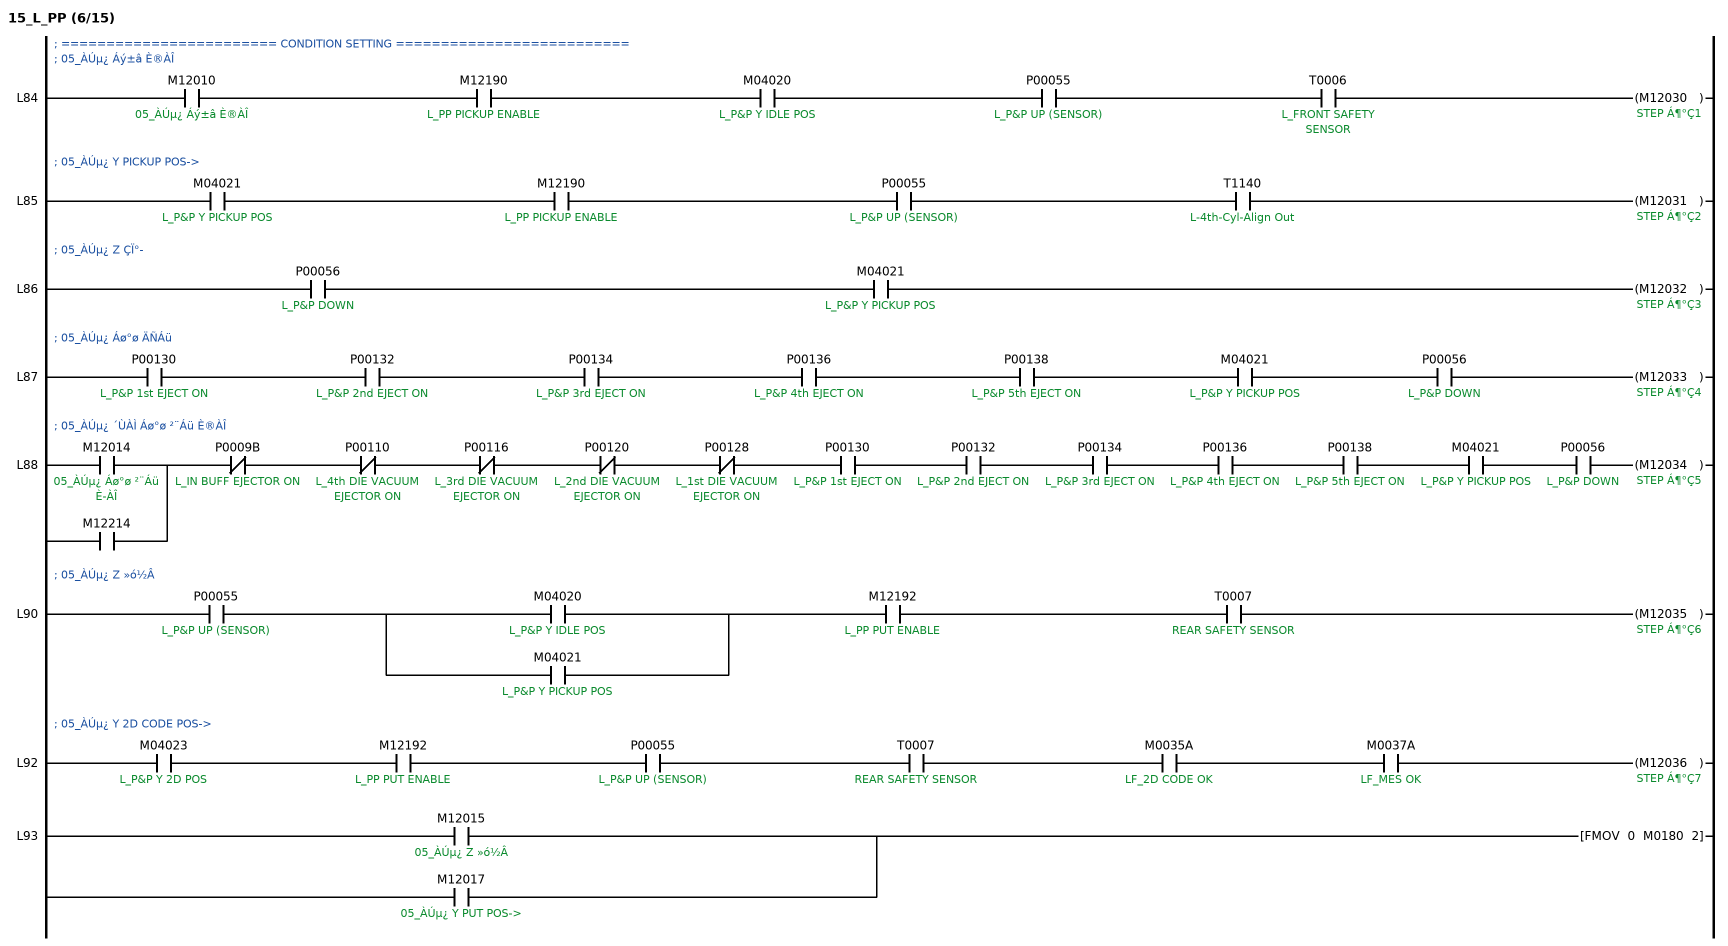
[picture p120: 15_L_PP rungs L84-L93]
// ======================== CONDITION SETTING ==========================
; L84
LOAD      M12010	// 05_ÀÚµ¿ Áý±â È®ÀÎ
AND       M12190	// L_PP PICKUP ENABLE
AND       M04020	// L_P&P Y IDLE POS
AND       P00055	// L_P&P UP (SENSOR)
AND       T0006	// L_FRONT SAFETY SENSOR
OUT       M12030	// STEP Á¶°Ç1
// output comment: 05_ÀÚµ¿ Áý±â È®ÀÎ
; L85
LOAD      M04021	// L_P&P Y PICKUP POS
AND       M12190	// L_PP PICKUP ENABLE
AND       P00055	// L_P&P UP (SENSOR)
AND       T1140	// L-4th-Cyl-Align Out
OUT       M12031	// STEP Á¶°Ç2
// output comment: 05_ÀÚµ¿ Y PICKUP POS->
; L86
LOAD      P00056	// L_P&P DOWN
AND       M04021	// L_P&P Y PICKUP POS
OUT       M12032	// STEP Á¶°Ç3
// output comment: 05_ÀÚµ¿ Z ÇÏ°­
; L87
LOAD      P00130	// L_P&P 1st EJECT ON
AND       P00132	// L_P&P 2nd EJECT ON
AND       P00134	// L_P&P 3rd EJECT ON
AND       P00136	// L_P&P 4th EJECT ON
AND       P00138	// L_P&P 5th EJECT ON
AND       M04021	// L_P&P Y PICKUP POS
AND       P00056	// L_P&P DOWN
OUT       M12033	// STEP Á¶°Ç4
// output comment: 05_ÀÚµ¿ Áø°ø ÄÑÁü
; L88
LOAD      M12014	// 05_ÀÚµ¿ Áø°ø ²¨Áü È­ÀÎ
OR        M12214
AND NOT   P0009B	// L_IN BUFF EJECTOR ON
AND NOT   P00110	// L_4th DIE VACUUM EJECTOR ON
AND NOT   P00116	// L_3rd DIE VACUUM EJECTOR ON
AND NOT   P00120	// L_2nd DIE VACUUM EJECTOR ON
AND NOT   P00128	// L_1st DIE VACUUM EJECTOR ON
AND       P00130	// L_P&P 1st EJECT ON
AND       P00132	// L_P&P 2nd EJECT ON
AND       P00134	// L_P&P 3rd EJECT ON
AND       P00136	// L_P&P 4th EJECT ON
AND       P00138	// L_P&P 5th EJECT ON
AND       M04021	// L_P&P Y PICKUP POS
AND       P00056	// L_P&P DOWN
OUT       M12034	// STEP Á¶°Ç5
// output comment: 05_ÀÚµ¿ ´ÙÀÌ Áø°ø ²¨Áü È®ÀÎ
; L90
LOAD      P00055	// L_P&P UP (SENSOR)
LOAD      M04020	// L_P&P Y IDLE POS
OR        M04021	// L_P&P Y PICKUP POS
AND LOAD
AND       M12192	// L_PP PUT ENABLE
AND       T0007	// REAR SAFETY SENSOR
OUT       M12035	// STEP Á¶°Ç6
// output comment: 05_ÀÚµ¿ Z »ó½Â
; L92
LOAD      M04023	// L_P&P Y 2D POS
AND       M12192	// L_PP PUT ENABLE
AND       P00055	// L_P&P UP (SENSOR)
AND       T0007	// REAR SAFETY SENSOR
AND       M0035A	// LF_2D CODE OK
AND       M0037A	// LF_MES OK
OUT       M12036	// STEP Á¶°Ç7
// output comment: 05_ÀÚµ¿ Y 2D CODE POS->
; L93
LOAD      M12015	// 05_ÀÚµ¿ Z »ó½Â
OR        M12017	// 05_ÀÚµ¿ Y PUT POS->
FMOV      0 M0180 2

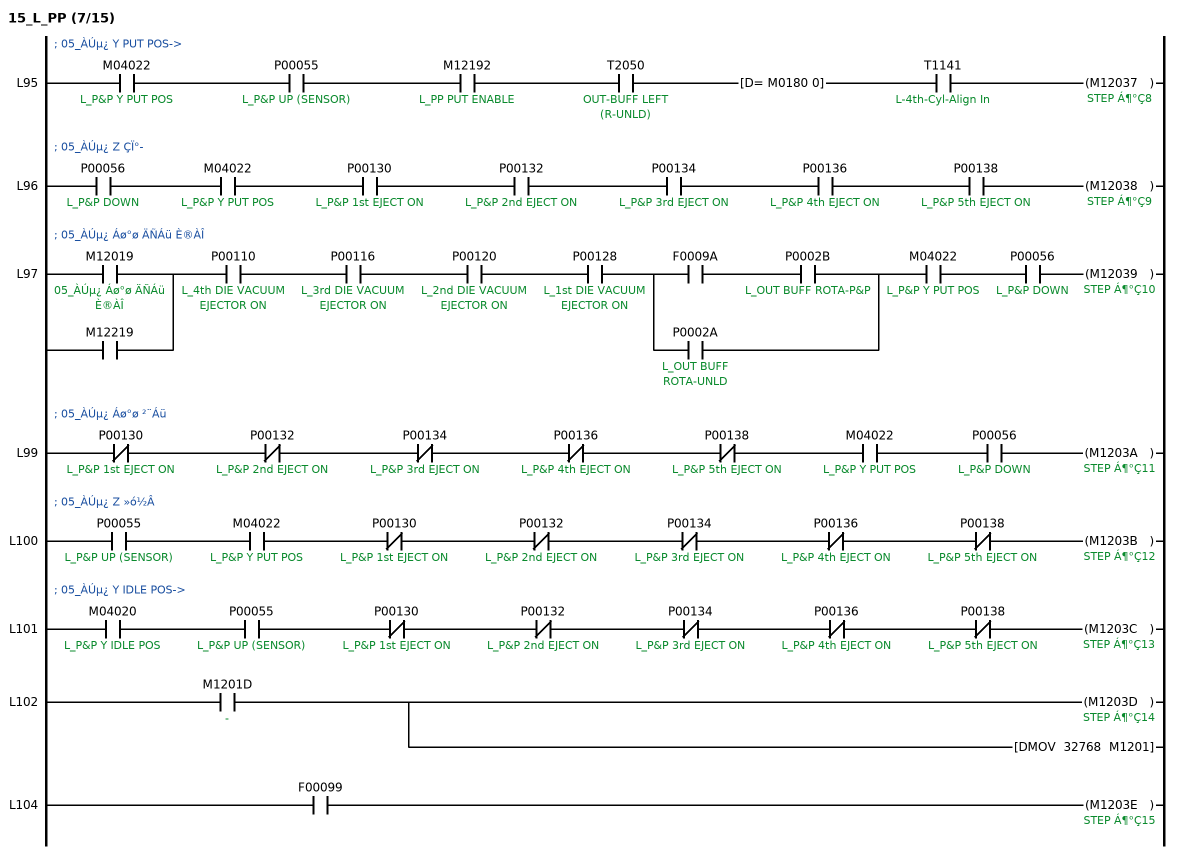
; L95
LOAD      M04022	// L_P&P Y PUT POS
AND       P00055	// L_P&P UP (SENSOR)
AND       M12192	// L_PP PUT ENABLE
AND       T2050	// OUT-BUFF LEFT (R-UNLD)
ANDD=     M0180 0
AND       T1141	// L-4th-Cyl-Align In
OUT       M12037	// STEP Á¶°Ç8
// output comment: 05_ÀÚµ¿ Y PUT POS->
; L96
LOAD      P00056	// L_P&P DOWN
AND       M04022	// L_P&P Y PUT POS
AND       P00130	// L_P&P 1st EJECT ON
AND       P00132	// L_P&P 2nd EJECT ON
AND       P00134	// L_P&P 3rd EJECT ON
AND       P00136	// L_P&P 4th EJECT ON
AND       P00138	// L_P&P 5th EJECT ON
OUT       M12038	// STEP Á¶°Ç9
// output comment: 05_ÀÚµ¿ Z ÇÏ°­
; L97
LOAD      M12019	// 05_ÀÚµ¿ Áø°ø ÄÑÁü È®ÀÎ
OR        M12219
AND       P00110	// L_4th DIE VACUUM EJECTOR ON
AND       P00116	// L_3rd DIE VACUUM EJECTOR ON
AND       P00120	// L_2nd DIE VACUUM EJECTOR ON
AND       P00128	// L_1st DIE VACUUM EJECTOR ON
LOAD      F0009A
AND       P0002B	// L_OUT BUFF ROTA-P&P
OR        P0002A	// L_OUT BUFF ROTA-UNLD
AND LOAD
AND       M04022	// L_P&P Y PUT POS
AND       P00056	// L_P&P DOWN
OUT       M12039	// STEP Á¶°Ç10
// output comment: 05_ÀÚµ¿ Áø°ø ÄÑÁü È®ÀÎ
; L99
LOAD NOT  P00130	// L_P&P 1st EJECT ON
AND NOT   P00132	// L_P&P 2nd EJECT ON
AND NOT   P00134	// L_P&P 3rd EJECT ON
AND NOT   P00136	// L_P&P 4th EJECT ON
AND NOT   P00138	// L_P&P 5th EJECT ON
AND       M04022	// L_P&P Y PUT POS
AND       P00056	// L_P&P DOWN
OUT       M1203A	// STEP Á¶°Ç11
// output comment: 05_ÀÚµ¿ Áø°ø ²¨Áü
; L100
LOAD      P00055	// L_P&P UP (SENSOR)
AND       M04022	// L_P&P Y PUT POS
AND NOT   P00130	// L_P&P 1st EJECT ON
AND NOT   P00132	// L_P&P 2nd EJECT ON
AND NOT   P00134	// L_P&P 3rd EJECT ON
AND NOT   P00136	// L_P&P 4th EJECT ON
AND NOT   P00138	// L_P&P 5th EJECT ON
OUT       M1203B	// STEP Á¶°Ç12
// output comment: 05_ÀÚµ¿ Z »ó½Â
; L101
LOAD      M04020	// L_P&P Y IDLE POS
AND       P00055	// L_P&P UP (SENSOR)
AND NOT   P00130	// L_P&P 1st EJECT ON
AND NOT   P00132	// L_P&P 2nd EJECT ON
AND NOT   P00134	// L_P&P 3rd EJECT ON
AND NOT   P00136	// L_P&P 4th EJECT ON
AND NOT   P00138	// L_P&P 5th EJECT ON
OUT       M1203C	// STEP Á¶°Ç13
// output comment: 05_ÀÚµ¿ Y IDLE POS->
; L102
LOAD      M1201D	// -
OUT       M1203D	// STEP Á¶°Ç14
DMOV      32768 M1201
; L104
LOAD      F00099
OUT       M1203E	// STEP Á¶°Ç15

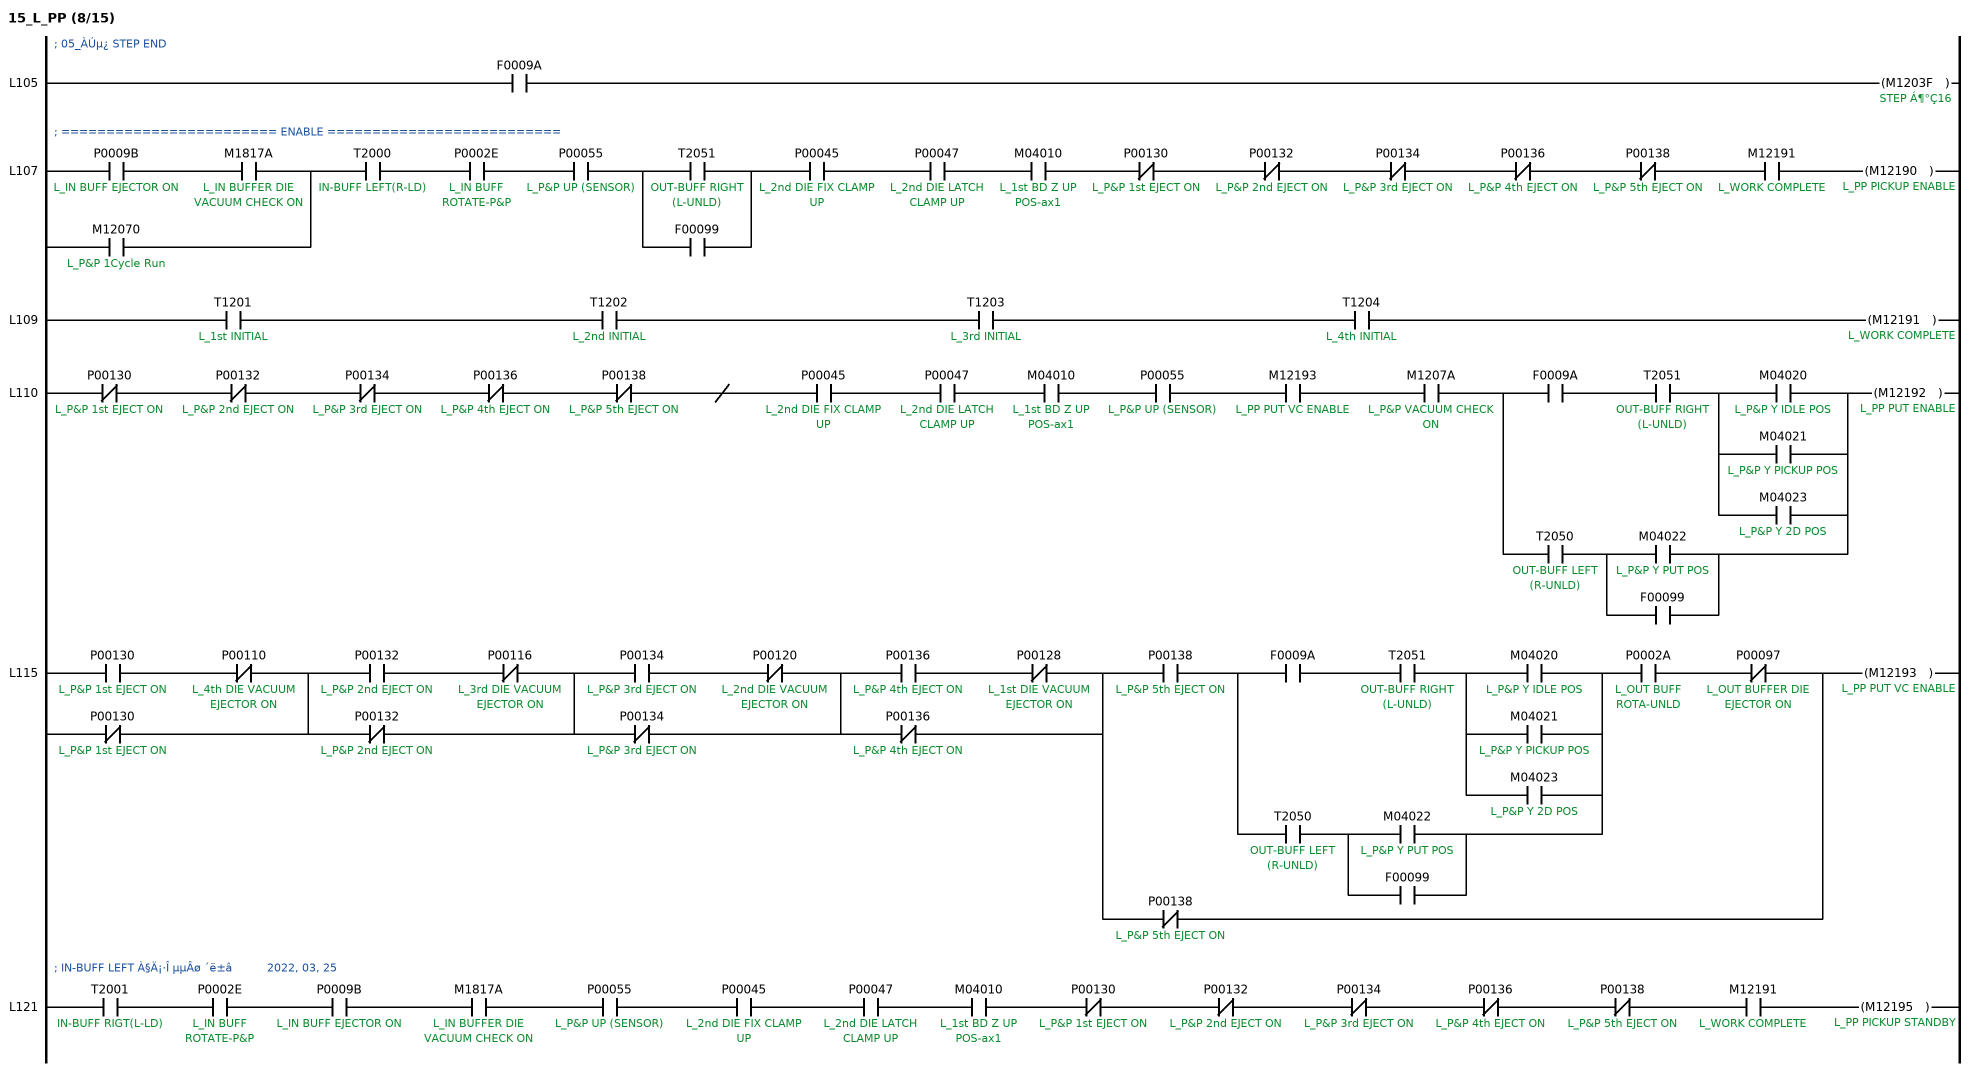
; L105
LOAD      F0009A
OUT       M1203F	// STEP Á¶°Ç16
// output comment: 05_ÀÚµ¿ STEP END
// ======================== ENABLE ==========================
; L107
LOAD      P0009B	// L_IN BUFF EJECTOR ON
AND       M1817A	// L_IN BUFFER DIE VACUUM CHECK ON
OR        M12070	// L_P&P 1Cycle Run
AND       T2000	// IN-BUFF LEFT(R-LD)
AND       P0002E	// L_IN BUFF ROTATE-P&P
AND       P00055	// L_P&P UP (SENSOR)
LOAD      T2051	// OUT-BUFF RIGHT (L-UNLD)
OR        F00099
AND LOAD
AND       P00045	// L_2nd DIE FIX CLAMP UP
AND       P00047	// L_2nd DIE LATCH CLAMP UP
AND       M04010	// L_1st BD Z UP POS-ax1
AND NOT   P00130	// L_P&P 1st EJECT ON
AND NOT   P00132	// L_P&P 2nd EJECT ON
AND NOT   P00134	// L_P&P 3rd EJECT ON
AND NOT   P00136	// L_P&P 4th EJECT ON
AND NOT   P00138	// L_P&P 5th EJECT ON
AND       M12191	// L_WORK COMPLETE
OUT       M12190	// L_PP PICKUP ENABLE
; L109
LOAD      T1201	// L_1st INITIAL
AND       T1202	// L_2nd INITIAL
AND       T1203	// L_3rd INITIAL
AND       T1204	// L_4th INITIAL
OUT       M12191	// L_WORK COMPLETE
; L110
LOAD NOT  P00130	// L_P&P 1st EJECT ON
AND NOT   P00132	// L_P&P 2nd EJECT ON
AND NOT   P00134	// L_P&P 3rd EJECT ON
AND NOT   P00136	// L_P&P 4th EJECT ON
AND NOT   P00138	// L_P&P 5th EJECT ON
NOT
AND       P00045	// L_2nd DIE FIX CLAMP UP
AND       P00047	// L_2nd DIE LATCH CLAMP UP
AND       M04010	// L_1st BD Z UP POS-ax1
AND       P00055	// L_P&P UP (SENSOR)
AND       M12193	// L_PP PUT VC ENABLE
AND       M1207A	// L_P&P VACUUM CHECK ON
LOAD      F0009A
AND       T2051	// OUT-BUFF RIGHT (L-UNLD)
LOAD      M04020	// L_P&P Y IDLE POS
OR        M04021	// L_P&P Y PICKUP POS
OR        M04023	// L_P&P Y 2D POS
AND LOAD
LOAD      T2050	// OUT-BUFF LEFT (R-UNLD)
LOAD      M04022	// L_P&P Y PUT POS
OR        F00099
AND LOAD
OR LOAD
AND LOAD
OUT       M12192	// L_PP PUT ENABLE
; L115
LOAD      P00130	// L_P&P 1st EJECT ON
AND NOT   P00110	// L_4th DIE VACUUM EJECTOR ON
OR NOT    P00130	// L_P&P 1st EJECT ON
LOAD      P00132	// L_P&P 2nd EJECT ON
AND NOT   P00116	// L_3rd DIE VACUUM EJECTOR ON
OR NOT    P00132	// L_P&P 2nd EJECT ON
AND LOAD
LOAD      P00134	// L_P&P 3rd EJECT ON
AND NOT   P00120	// L_2nd DIE VACUUM EJECTOR ON
OR NOT    P00134	// L_P&P 3rd EJECT ON
AND LOAD
LOAD      P00136	// L_P&P 4th EJECT ON
AND NOT   P00128	// L_1st DIE VACUUM EJECTOR ON
OR NOT    P00136	// L_P&P 4th EJECT ON
AND LOAD
LOAD      P00138	// L_P&P 5th EJECT ON
LOAD      F0009A
AND       T2051	// OUT-BUFF RIGHT (L-UNLD)
LOAD      M04020	// L_P&P Y IDLE POS
OR        M04021	// L_P&P Y PICKUP POS
OR        M04023	// L_P&P Y 2D POS
AND LOAD
LOAD      T2050	// OUT-BUFF LEFT (R-UNLD)
LOAD      M04022	// L_P&P Y PUT POS
OR        F00099
AND LOAD
OR LOAD
AND LOAD
AND       P0002A	// L_OUT BUFF ROTA-UNLD
AND NOT   P00097	// L_OUT BUFFER DIE EJECTOR ON
OR NOT    P00138	// L_P&P 5th EJECT ON
AND LOAD
OUT       M12193	// L_PP PUT VC ENABLE
; L121
LOAD      T2001	// IN-BUFF RIGT(L-LD)
AND       P0002E	// L_IN BUFF ROTATE-P&P
AND       P0009B	// L_IN BUFF EJECTOR ON
AND       M1817A	// L_IN BUFFER DIE VACUUM CHECK ON
AND       P00055	// L_P&P UP (SENSOR)
AND       P00045	// L_2nd DIE FIX CLAMP UP
AND       P00047	// L_2nd DIE LATCH CLAMP UP
AND       M04010	// L_1st BD Z UP POS-ax1
AND NOT   P00130	// L_P&P 1st EJECT ON
AND NOT   P00132	// L_P&P 2nd EJECT ON
AND NOT   P00134	// L_P&P 3rd EJECT ON
AND NOT   P00136	// L_P&P 4th EJECT ON
AND NOT   P00138	// L_P&P 5th EJECT ON
AND       M12191	// L_WORK COMPLETE
OUT       M12195	// L_PP PICKUP STANDBY
// output comment: IN-BUFF LEFT À§Ä¡·Î µµÂø ´ë±â          2022, 03, 25

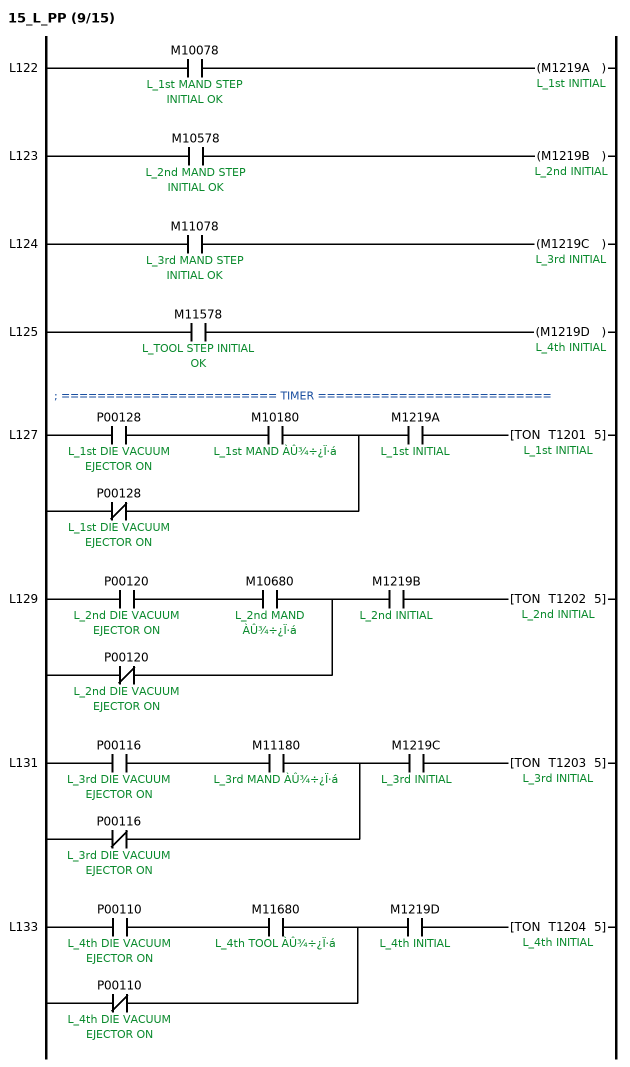
; L122
LOAD      M10078	// L_1st MAND STEP INITIAL OK
OUT       M1219A	// L_1st INITIAL
; L123
LOAD      M10578	// L_2nd MAND STEP INITIAL OK
OUT       M1219B	// L_2nd INITIAL
; L124
LOAD      M11078	// L_3rd MAND STEP INITIAL OK
OUT       M1219C	// L_3rd INITIAL
; L125
LOAD      M11578	// L_TOOL STEP INITIAL OK
OUT       M1219D	// L_4th INITIAL
// ======================== TIMER ==========================
; L127
LOAD      P00128	// L_1st DIE VACUUM EJECTOR ON
AND       M10180	// L_1st MAND ÀÛ¾÷¿Ï·á
OR NOT    P00128	// L_1st DIE VACUUM EJECTOR ON
AND       M1219A	// L_1st INITIAL
TON       T1201 5	// L_1st INITIAL
; L129
LOAD      P00120	// L_2nd DIE VACUUM EJECTOR ON
AND       M10680	// L_2nd MAND ÀÛ¾÷¿Ï·á
OR NOT    P00120	// L_2nd DIE VACUUM EJECTOR ON
AND       M1219B	// L_2nd INITIAL
TON       T1202 5	// L_2nd INITIAL
; L131
LOAD      P00116	// L_3rd DIE VACUUM EJECTOR ON
AND       M11180	// L_3rd MAND ÀÛ¾÷¿Ï·á
OR NOT    P00116	// L_3rd DIE VACUUM EJECTOR ON
AND       M1219C	// L_3rd INITIAL
TON       T1203 5	// L_3rd INITIAL
; L133
LOAD      P00110	// L_4th DIE VACUUM EJECTOR ON
AND       M11680	// L_4th TOOL ÀÛ¾÷¿Ï·á
OR NOT    P00110	// L_4th DIE VACUUM EJECTOR ON
AND       M1219D	// L_4th INITIAL
TON       T1204 5	// L_4th INITIAL

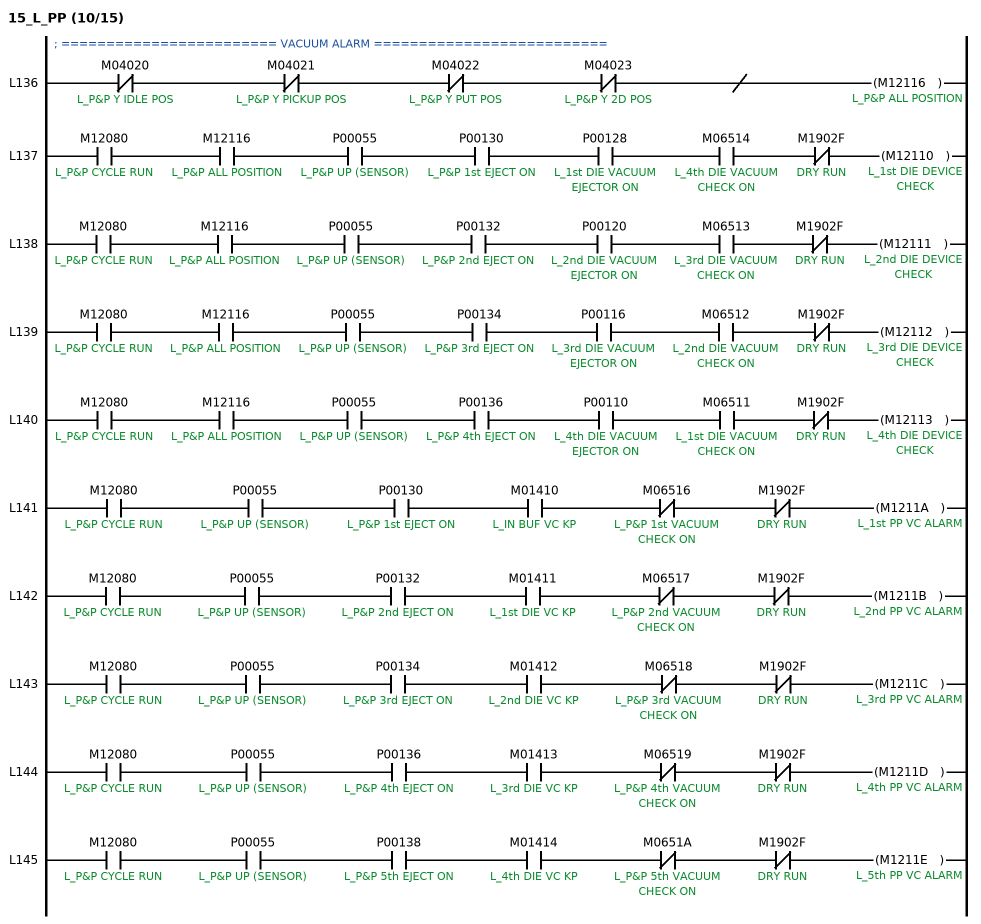
// ======================== VACUUM ALARM ==========================
; L136
LOAD NOT  M04020	// L_P&P Y IDLE POS
AND NOT   M04021	// L_P&P Y PICKUP POS
AND NOT   M04022	// L_P&P Y PUT POS
AND NOT   M04023	// L_P&P Y 2D POS
NOT
OUT       M12116	// L_P&P ALL POSITION
; L137
LOAD      M12080	// L_P&P CYCLE RUN
AND       M12116	// L_P&P ALL POSITION
AND       P00055	// L_P&P UP (SENSOR)
AND       P00130	// L_P&P 1st EJECT ON
AND       P00128	// L_1st DIE VACUUM EJECTOR ON
AND       M06514	// L_4th DIE VACUUM CHECK ON
AND NOT   M1902F	// DRY RUN
OUT       M12110	// L_1st DIE DEVICE CHECK
; L138
LOAD      M12080	// L_P&P CYCLE RUN
AND       M12116	// L_P&P ALL POSITION
AND       P00055	// L_P&P UP (SENSOR)
AND       P00132	// L_P&P 2nd EJECT ON
AND       P00120	// L_2nd DIE VACUUM EJECTOR ON
AND       M06513	// L_3rd DIE VACUUM CHECK ON
AND NOT   M1902F	// DRY RUN
OUT       M12111	// L_2nd DIE DEVICE CHECK
; L139
LOAD      M12080	// L_P&P CYCLE RUN
AND       M12116	// L_P&P ALL POSITION
AND       P00055	// L_P&P UP (SENSOR)
AND       P00134	// L_P&P 3rd EJECT ON
AND       P00116	// L_3rd DIE VACUUM EJECTOR ON
AND       M06512	// L_2nd DIE VACUUM CHECK ON
AND NOT   M1902F	// DRY RUN
OUT       M12112	// L_3rd DIE DEVICE CHECK
; L140
LOAD      M12080	// L_P&P CYCLE RUN
AND       M12116	// L_P&P ALL POSITION
AND       P00055	// L_P&P UP (SENSOR)
AND       P00136	// L_P&P 4th EJECT ON
AND       P00110	// L_4th DIE VACUUM EJECTOR ON
AND       M06511	// L_1st DIE VACUUM CHECK ON
AND NOT   M1902F	// DRY RUN
OUT       M12113	// L_4th DIE DEVICE CHECK
; L141
LOAD      M12080	// L_P&P CYCLE RUN
AND       P00055	// L_P&P UP (SENSOR)
AND       P00130	// L_P&P 1st EJECT ON
AND       M01410	// L_IN BUF VC KP
AND NOT   M06516	// L_P&P 1st VACUUM CHECK ON
AND NOT   M1902F	// DRY RUN
OUT       M1211A	// L_1st PP VC ALARM
; L142
LOAD      M12080	// L_P&P CYCLE RUN
AND       P00055	// L_P&P UP (SENSOR)
AND       P00132	// L_P&P 2nd EJECT ON
AND       M01411	// L_1st DIE VC KP
AND NOT   M06517	// L_P&P 2nd VACUUM CHECK ON
AND NOT   M1902F	// DRY RUN
OUT       M1211B	// L_2nd PP VC ALARM
; L143
LOAD      M12080	// L_P&P CYCLE RUN
AND       P00055	// L_P&P UP (SENSOR)
AND       P00134	// L_P&P 3rd EJECT ON
AND       M01412	// L_2nd DIE VC KP
AND NOT   M06518	// L_P&P 3rd VACUUM CHECK ON
AND NOT   M1902F	// DRY RUN
OUT       M1211C	// L_3rd PP VC ALARM
; L144
LOAD      M12080	// L_P&P CYCLE RUN
AND       P00055	// L_P&P UP (SENSOR)
AND       P00136	// L_P&P 4th EJECT ON
AND       M01413	// L_3rd DIE VC KP
AND NOT   M06519	// L_P&P 4th VACUUM CHECK ON
AND NOT   M1902F	// DRY RUN
OUT       M1211D	// L_4th PP VC ALARM
; L145
LOAD      M12080	// L_P&P CYCLE RUN
AND       P00055	// L_P&P UP (SENSOR)
AND       P00138	// L_P&P 5th EJECT ON
AND       M01414	// L_4th DIE VC KP
AND NOT   M0651A	// L_P&P 5th VACUUM CHECK ON
AND NOT   M1902F	// DRY RUN
OUT       M1211E	// L_5th PP VC ALARM

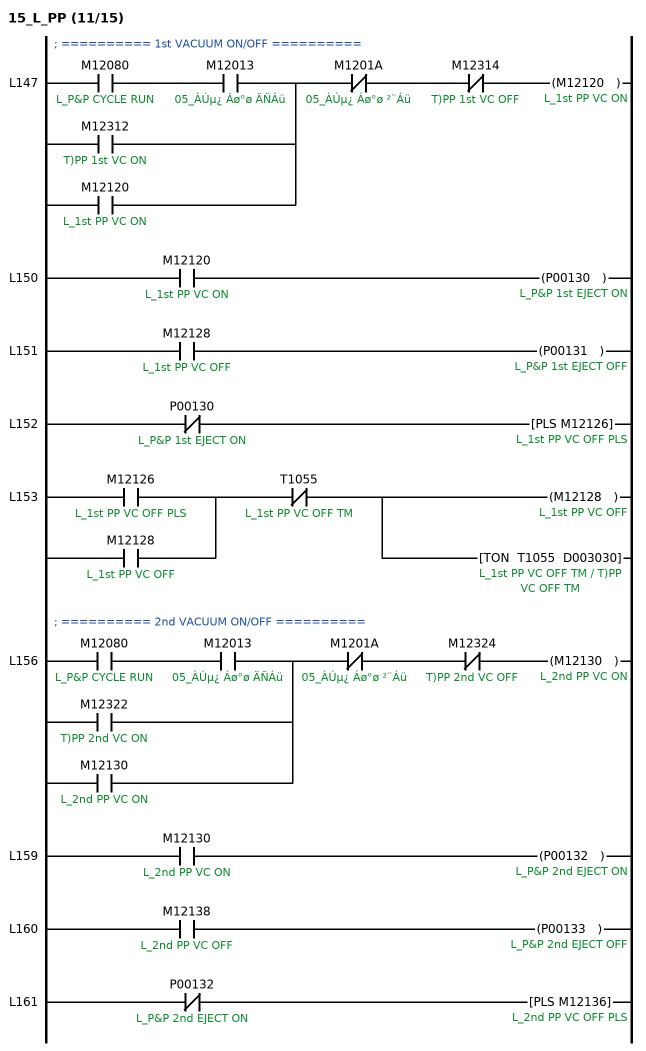
// ========== 1st VACUUM ON/OFF ==========
; L147
LOAD      M12080	// L_P&P CYCLE RUN
AND       M12013	// 05_ÀÚµ¿ Áø°ø ÄÑÁü
OR        M12312	// T)PP 1st VC ON
OR        M12120	// L_1st PP VC ON
AND NOT   M1201A	// 05_ÀÚµ¿ Áø°ø ²¨Áü
AND NOT   M12314	// T)PP 1st VC OFF
OUT       M12120	// L_1st PP VC ON
; L150
LOAD      M12120	// L_1st PP VC ON
OUT       P00130	// L_P&P 1st EJECT ON
; L151
LOAD      M12128	// L_1st PP VC OFF
OUT       P00131	// L_P&P 1st EJECT OFF
; L152
LOAD NOT  P00130	// L_P&P 1st EJECT ON
OUTP      M12126	// L_1st PP VC OFF PLS
; L153
LOAD      M12126	// L_1st PP VC OFF PLS
OR        M12128	// L_1st PP VC OFF
AND NOT   T1055	// L_1st PP VC OFF TM
OUT       M12128	// L_1st PP VC OFF
TON       T1055 D003030	// L_1st PP VC OFF TM / T)PP VC OFF TM
// ========== 2nd VACUUM ON/OFF ==========
; L156
LOAD      M12080	// L_P&P CYCLE RUN
AND       M12013	// 05_ÀÚµ¿ Áø°ø ÄÑÁü
OR        M12322	// T)PP 2nd VC ON
OR        M12130	// L_2nd PP VC ON
AND NOT   M1201A	// 05_ÀÚµ¿ Áø°ø ²¨Áü
AND NOT   M12324	// T)PP 2nd VC OFF
OUT       M12130	// L_2nd PP VC ON
; L159
LOAD      M12130	// L_2nd PP VC ON
OUT       P00132	// L_P&P 2nd EJECT ON
; L160
LOAD      M12138	// L_2nd PP VC OFF
OUT       P00133	// L_P&P 2nd EJECT OFF
; L161
LOAD NOT  P00132	// L_P&P 2nd EJECT ON
OUTP      M12136	// L_2nd PP VC OFF PLS

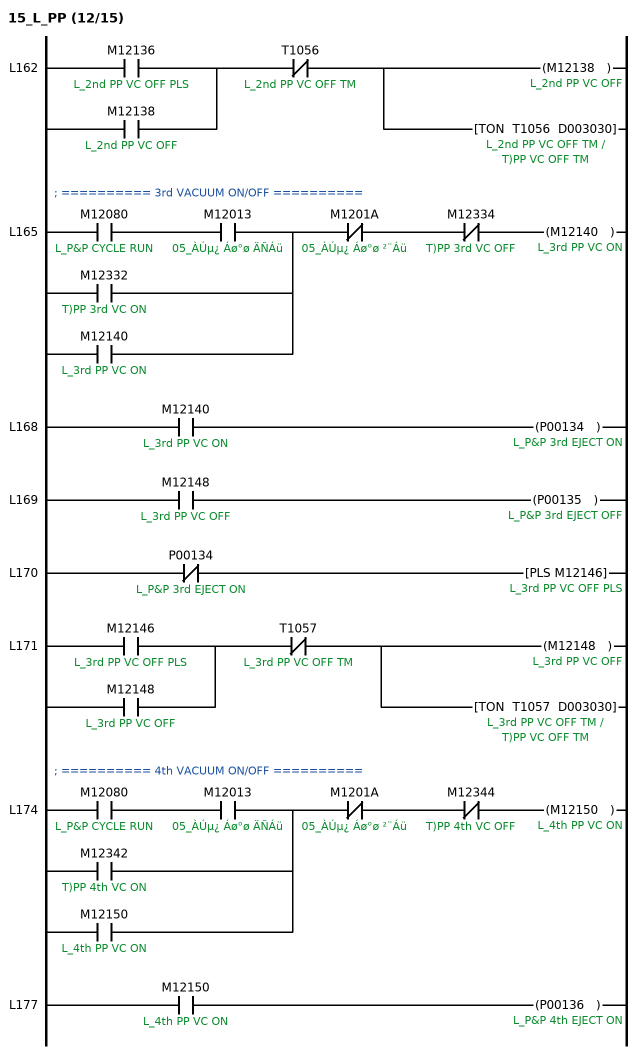
; L162
LOAD      M12136	// L_2nd PP VC OFF PLS
OR        M12138	// L_2nd PP VC OFF
AND NOT   T1056	// L_2nd PP VC OFF TM
OUT       M12138	// L_2nd PP VC OFF
TON       T1056 D003030	// L_2nd PP VC OFF TM / T)PP VC OFF TM
// ========== 3rd VACUUM ON/OFF ==========
; L165
LOAD      M12080	// L_P&P CYCLE RUN
AND       M12013	// 05_ÀÚµ¿ Áø°ø ÄÑÁü
OR        M12332	// T)PP 3rd VC ON
OR        M12140	// L_3rd PP VC ON
AND NOT   M1201A	// 05_ÀÚµ¿ Áø°ø ²¨Áü
AND NOT   M12334	// T)PP 3rd VC OFF
OUT       M12140	// L_3rd PP VC ON
; L168
LOAD      M12140	// L_3rd PP VC ON
OUT       P00134	// L_P&P 3rd EJECT ON
; L169
LOAD      M12148	// L_3rd PP VC OFF
OUT       P00135	// L_P&P 3rd EJECT OFF
; L170
LOAD NOT  P00134	// L_P&P 3rd EJECT ON
OUTP      M12146	// L_3rd PP VC OFF PLS
; L171
LOAD      M12146	// L_3rd PP VC OFF PLS
OR        M12148	// L_3rd PP VC OFF
AND NOT   T1057	// L_3rd PP VC OFF TM
OUT       M12148	// L_3rd PP VC OFF
TON       T1057 D003030	// L_3rd PP VC OFF TM / T)PP VC OFF TM
// ========== 4th VACUUM ON/OFF ==========
; L174
LOAD      M12080	// L_P&P CYCLE RUN
AND       M12013	// 05_ÀÚµ¿ Áø°ø ÄÑÁü
OR        M12342	// T)PP 4th VC ON
OR        M12150	// L_4th PP VC ON
AND NOT   M1201A	// 05_ÀÚµ¿ Áø°ø ²¨Áü
AND NOT   M12344	// T)PP 4th VC OFF
OUT       M12150	// L_4th PP VC ON
; L177
LOAD      M12150	// L_4th PP VC ON
OUT       P00136	// L_P&P 4th EJECT ON

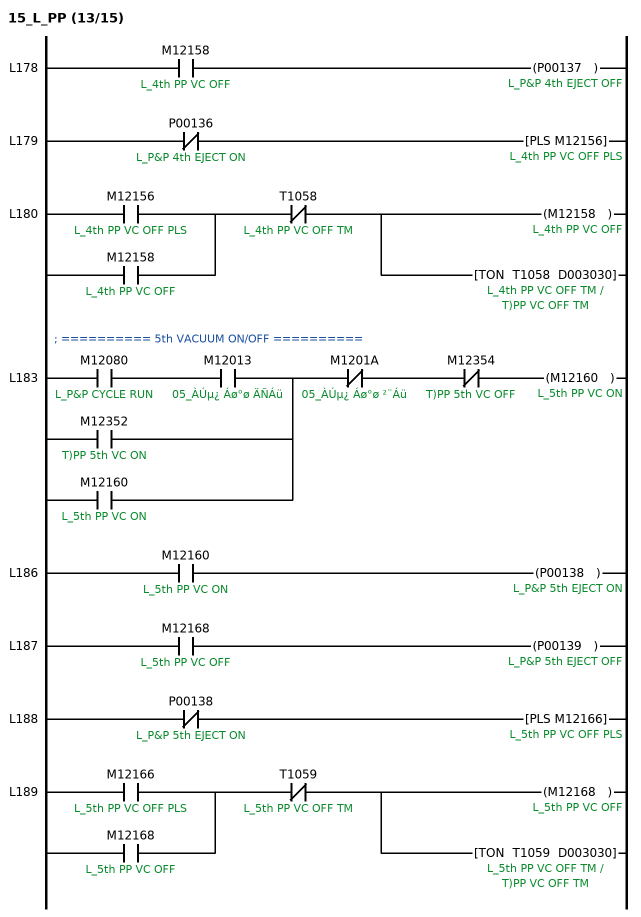
; L178
LOAD      M12158	// L_4th PP VC OFF
OUT       P00137	// L_P&P 4th EJECT OFF
; L179
LOAD NOT  P00136	// L_P&P 4th EJECT ON
OUTP      M12156	// L_4th PP VC OFF PLS
; L180
LOAD      M12156	// L_4th PP VC OFF PLS
OR        M12158	// L_4th PP VC OFF
AND NOT   T1058	// L_4th PP VC OFF TM
OUT       M12158	// L_4th PP VC OFF
TON       T1058 D003030	// L_4th PP VC OFF TM / T)PP VC OFF TM
// ========== 5th VACUUM ON/OFF ==========
; L183
LOAD      M12080	// L_P&P CYCLE RUN
AND       M12013	// 05_ÀÚµ¿ Áø°ø ÄÑÁü
OR        M12352	// T)PP 5th VC ON
OR        M12160	// L_5th PP VC ON
AND NOT   M1201A	// 05_ÀÚµ¿ Áø°ø ²¨Áü
AND NOT   M12354	// T)PP 5th VC OFF
OUT       M12160	// L_5th PP VC ON
; L186
LOAD      M12160	// L_5th PP VC ON
OUT       P00138	// L_P&P 5th EJECT ON
; L187
LOAD      M12168	// L_5th PP VC OFF
OUT       P00139	// L_P&P 5th EJECT OFF
; L188
LOAD NOT  P00138	// L_P&P 5th EJECT ON
OUTP      M12166	// L_5th PP VC OFF PLS
; L189
LOAD      M12166	// L_5th PP VC OFF PLS
OR        M12168	// L_5th PP VC OFF
AND NOT   T1059	// L_5th PP VC OFF TM
OUT       M12168	// L_5th PP VC OFF
TON       T1059 D003030	// L_5th PP VC OFF TM / T)PP VC OFF TM

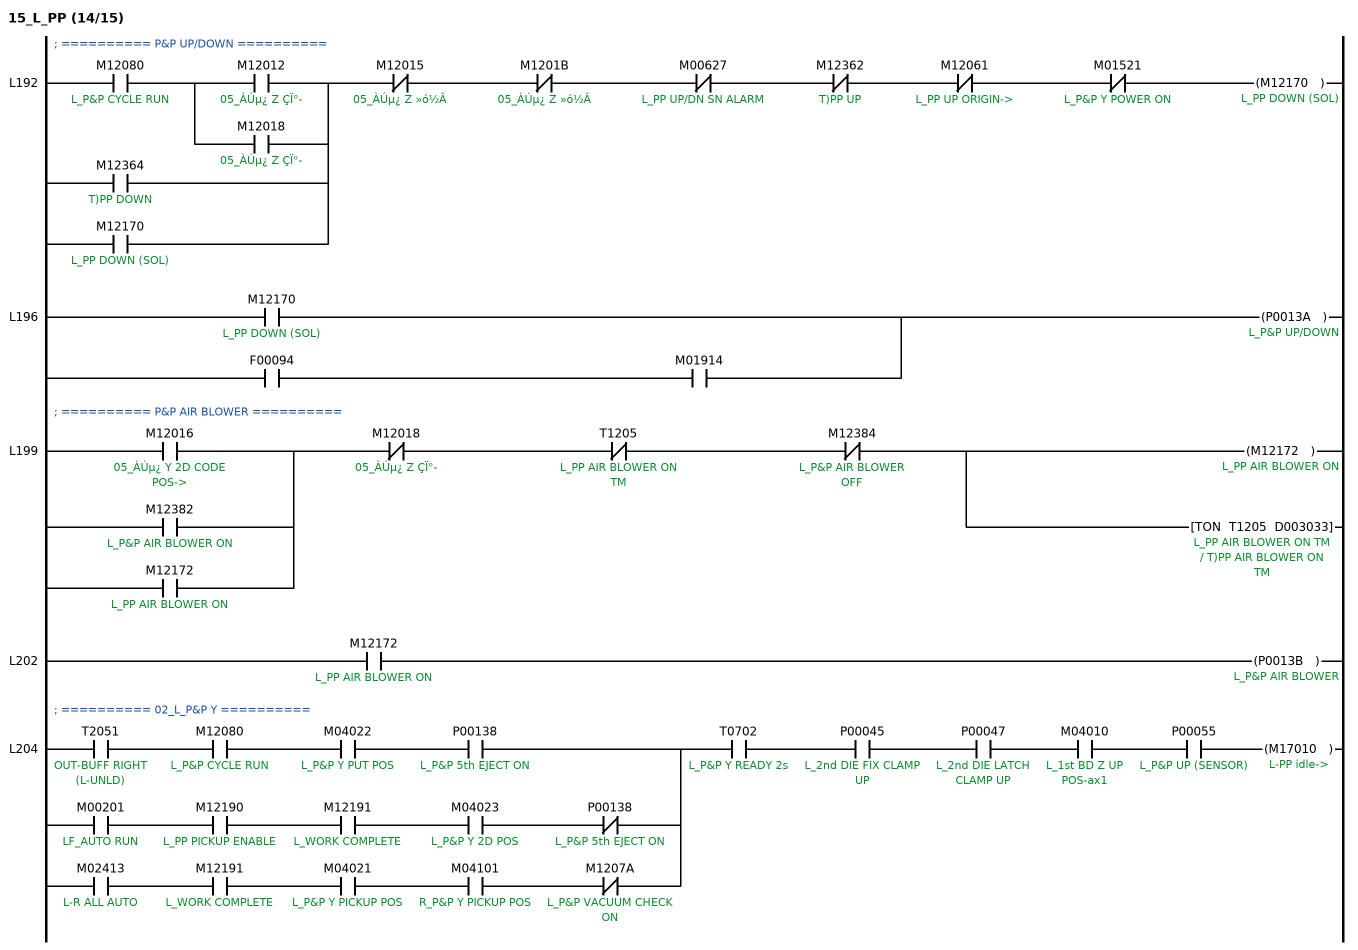
// ========== P&P UP/DOWN ==========
; L192
LOAD      M12080	// L_P&P CYCLE RUN
LOAD      M12012	// 05_ÀÚµ¿ Z ÇÏ°­
OR        M12018	// 05_ÀÚµ¿ Z ÇÏ°­
AND LOAD
OR        M12364	// T)PP DOWN
OR        M12170	// L_PP DOWN (SOL)
AND NOT   M12015	// 05_ÀÚµ¿ Z »ó½Â
AND NOT   M1201B	// 05_ÀÚµ¿ Z »ó½Â
AND NOT   M00627	// L_PP UP/DN SN ALARM
AND NOT   M12362	// T)PP UP
AND NOT   M12061	// L_PP UP ORIGIN->
AND NOT   M01521	// L_P&P Y POWER ON
OUT       M12170	// L_PP DOWN (SOL)
; L196
LOAD      M12170	// L_PP DOWN (SOL)
LOAD      F00094
AND       M01914
OR LOAD
OUT       P0013A	// L_P&P UP/DOWN
// ========== P&P AIR BLOWER ==========
; L199
LOAD      M12016	// 05_ÀÚµ¿ Y 2D CODE POS->
OR        M12382	// L_P&P AIR BLOWER ON
OR        M12172	// L_PP AIR BLOWER ON
AND NOT   M12018	// 05_ÀÚµ¿ Z ÇÏ°­
AND NOT   T1205	// L_PP AIR BLOWER ON TM
AND NOT   M12384	// L_P&P AIR BLOWER OFF
OUT       M12172	// L_PP AIR BLOWER ON
TON       T1205 D003033	// L_PP AIR BLOWER ON TM / T)PP AIR BLOWER ON TM
; L202
LOAD      M12172	// L_PP AIR BLOWER ON
OUT       P0013B	// L_P&P AIR BLOWER
// ========== 02_L_P&P Y ==========
; L204
LOAD      T2051	// OUT-BUFF RIGHT (L-UNLD)
AND       M12080	// L_P&P CYCLE RUN
AND       M04022	// L_P&P Y PUT POS
AND       P00138	// L_P&P 5th EJECT ON
LOAD      M00201	// LF_AUTO RUN
AND       M12190	// L_PP PICKUP ENABLE
AND       M12191	// L_WORK COMPLETE
AND       M04023	// L_P&P Y 2D POS
AND NOT   P00138	// L_P&P 5th EJECT ON
OR LOAD
LOAD      M02413	// L-R ALL AUTO
AND       M12191	// L_WORK COMPLETE
AND       M04021	// L_P&P Y PICKUP POS
AND       M04101	// R_P&P Y PICKUP POS
AND NOT   M1207A	// L_P&P VACUUM CHECK ON
OR LOAD
AND       T0702	// L_P&P Y READY 2s
AND       P00045	// L_2nd DIE FIX CLAMP UP
AND       P00047	// L_2nd DIE LATCH CLAMP UP
AND       M04010	// L_1st BD Z UP POS-ax1
AND       P00055	// L_P&P UP (SENSOR)
OUT       M17010	// L-PP idle->

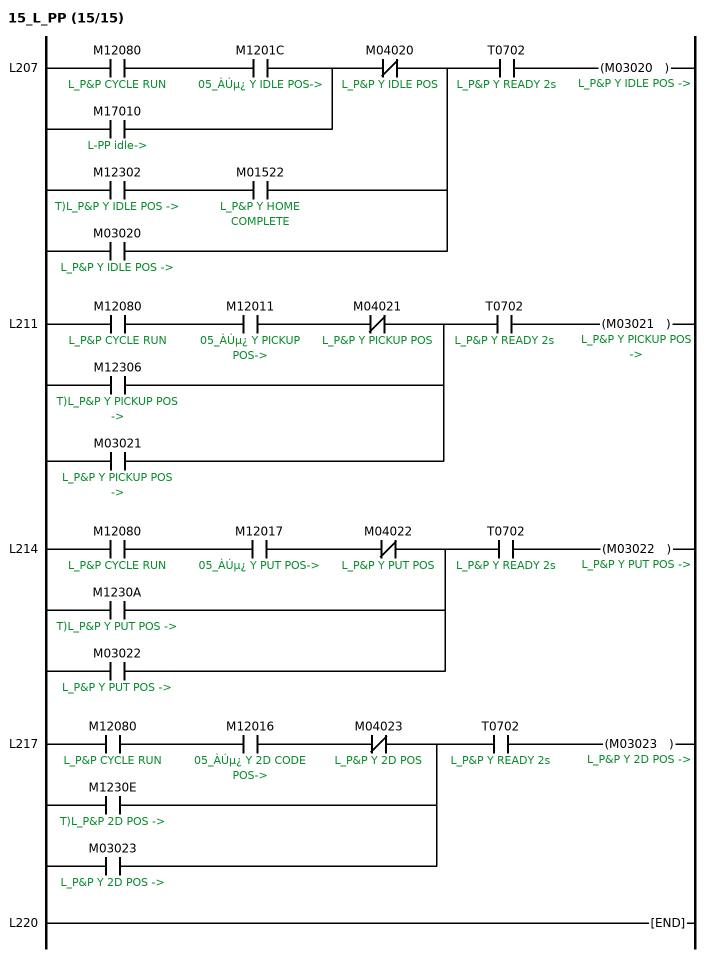
; L207
LOAD      M12080	// L_P&P CYCLE RUN
AND       M1201C	// 05_ÀÚµ¿ Y IDLE POS->
OR        M17010	// L-PP idle->
AND NOT   M04020	// L_P&P Y IDLE POS
LOAD      M12302	// T)L_P&P Y IDLE POS ->
AND       M01522	// L_P&P Y HOME COMPLETE
OR LOAD
OR        M03020	// L_P&P Y IDLE POS ->
AND       T0702	// L_P&P Y READY 2s
OUT       M03020	// L_P&P Y IDLE POS ->
; L211
LOAD      M12080	// L_P&P CYCLE RUN
AND       M12011	// 05_ÀÚµ¿ Y PICKUP POS->
AND NOT   M04021	// L_P&P Y PICKUP POS
OR        M12306	// T)L_P&P Y PICKUP POS ->
OR        M03021	// L_P&P Y PICKUP POS ->
AND       T0702	// L_P&P Y READY 2s
OUT       M03021	// L_P&P Y PICKUP POS ->
; L214
LOAD      M12080	// L_P&P CYCLE RUN
AND       M12017	// 05_ÀÚµ¿ Y PUT POS->
AND NOT   M04022	// L_P&P Y PUT POS
OR        M1230A	// T)L_P&P Y PUT POS ->
OR        M03022	// L_P&P Y PUT POS ->
AND       T0702	// L_P&P Y READY 2s
OUT       M03022	// L_P&P Y PUT POS ->
; L217
LOAD      M12080	// L_P&P CYCLE RUN
AND       M12016	// 05_ÀÚµ¿ Y 2D CODE POS->
AND NOT   M04023	// L_P&P Y 2D POS
OR        M1230E	// T)L_P&P 2D POS ->
OR        M03023	// L_P&P Y 2D POS ->
AND       T0702	// L_P&P Y READY 2s
OUT       M03023	// L_P&P Y 2D POS ->
; L220
END

PROGRAM 16_R_1st_MAND (task: ½ºÄµ ÇÁ·Î±×·¥)

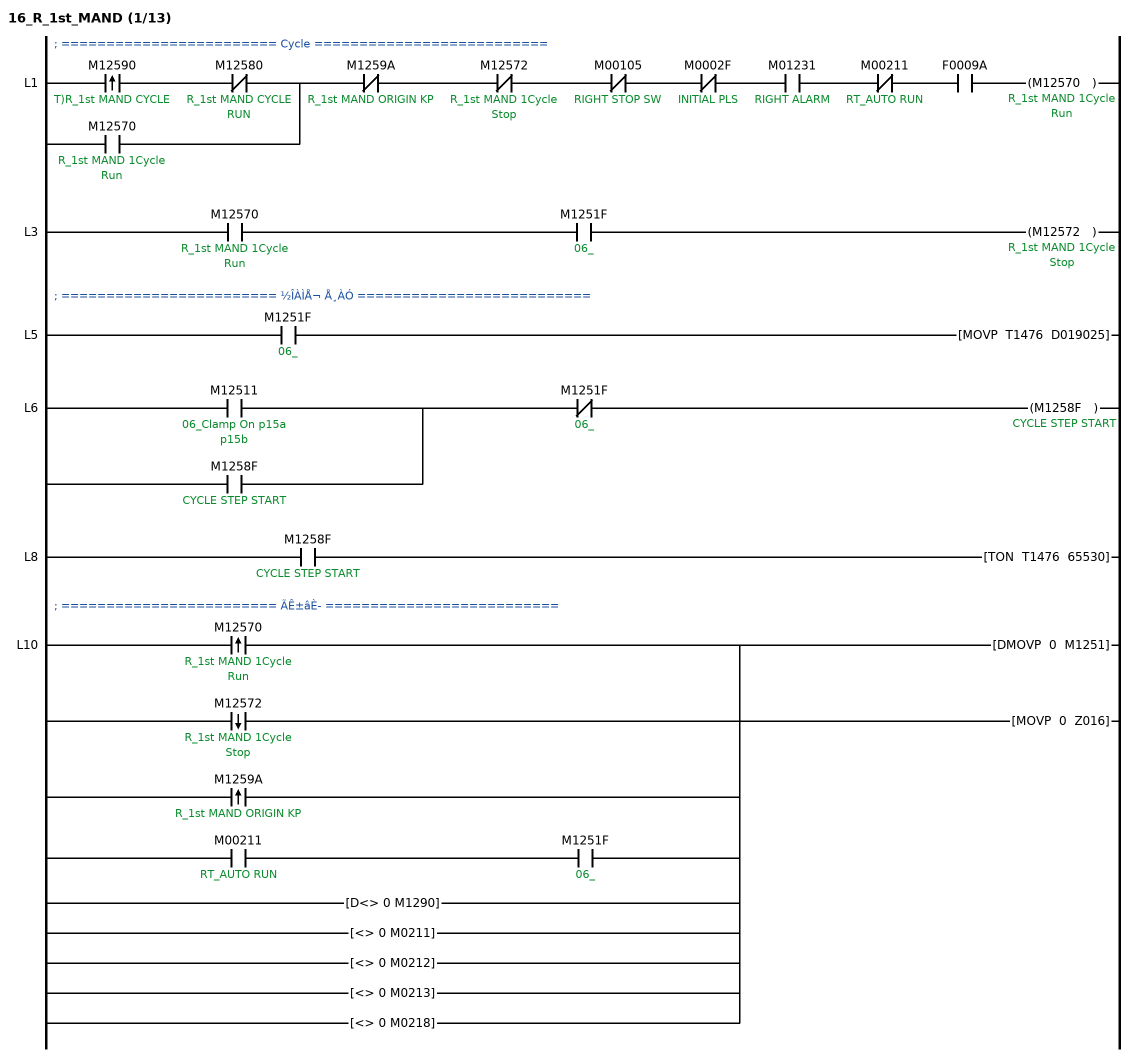
// ======================== Cycle ==========================
; L1
LOADP     M12590	// T)R_1st MAND CYCLE
AND NOT   M12580	// R_1st MAND CYCLE RUN
OR        M12570	// R_1st MAND 1Cycle Run
AND NOT   M1259A	// R_1st MAND ORIGIN KP
AND NOT   M12572	// R_1st MAND 1Cycle Stop
AND NOT   M00105	// RIGHT STOP SW
AND NOT   M0002F	// INITIAL PLS
AND       M01231	// RIGHT ALARM
AND NOT   M00211	// RT_AUTO RUN
AND       F0009A
OUT       M12570	// R_1st MAND 1Cycle Run
; L3
LOAD      M12570	// R_1st MAND 1Cycle Run
AND       M1251F	// 06_
OUT       M12572	// R_1st MAND 1Cycle Stop
// ======================== ½ÎÀÌÅ¬ Å¸ÀÓ ==========================
; L5
LOAD      M1251F	// 06_
MOVP      T1476 D019025
; L6
LOAD      M12511	// 06_Clamp On p15a p15b
OR        M1258F	// CYCLE STEP START
AND NOT   M1251F	// 06_
OUT       M1258F	// CYCLE STEP START
; L8
LOAD      M1258F	// CYCLE STEP START
TON       T1476 65530
// ======================== ÃÊ±âÈ­ ==========================
; L10
LOADP     M12570	// R_1st MAND 1Cycle Run
ORN       M12572	// R_1st MAND 1Cycle Stop
ORP       M1259A	// R_1st MAND ORIGIN KP
LOAD      M00211	// RT_AUTO RUN
AND       M1251F	// 06_
OR LOAD
ORD<>     0 M1290
OR<>      0 M0211
OR<>      0 M0212
OR<>      0 M0213
OR<>      0 M0218
DMOVP     0 M1251
MOVP      0 Z016

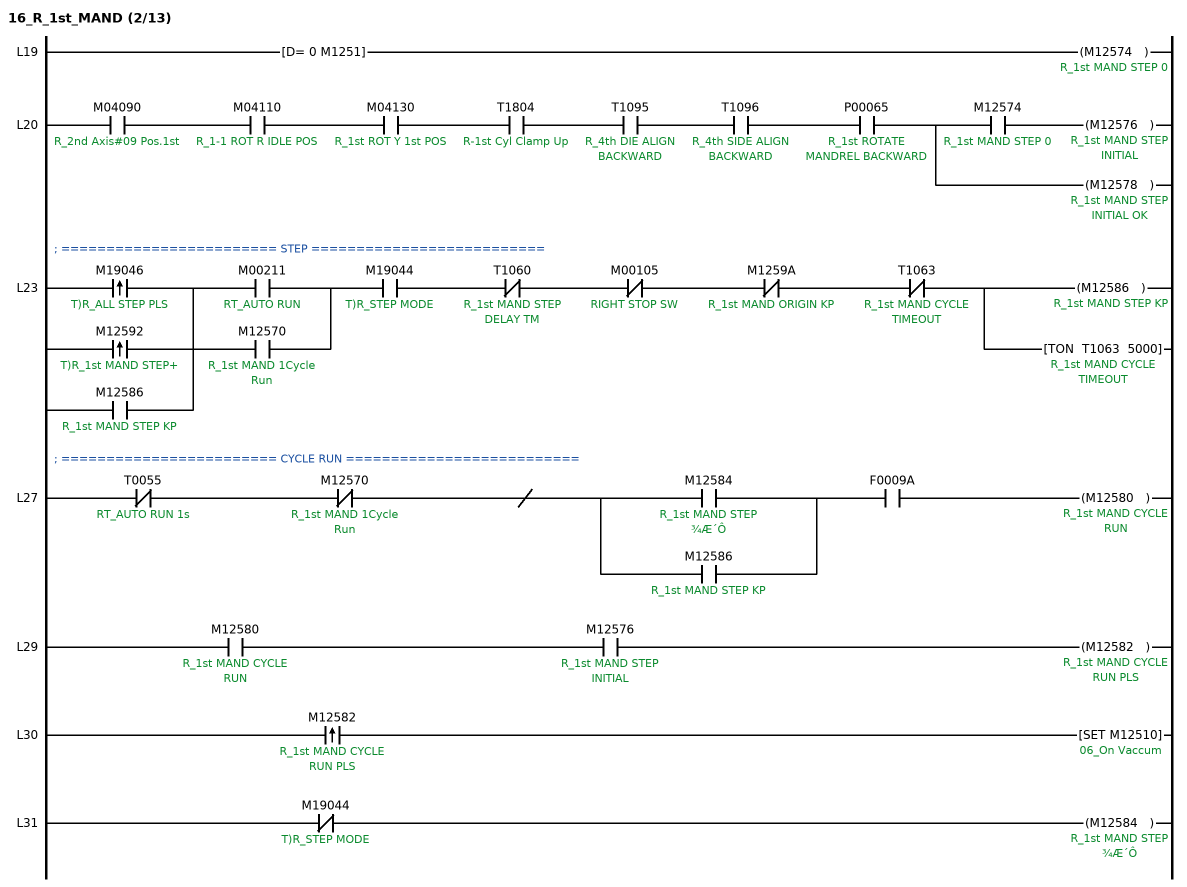
; L19
LOADD=    0 M1251
OUT       M12574	// R_1st MAND STEP 0
; L20
LOAD      M04090	// R_2nd Axis#09 Pos.1st
AND       M04110	// R_1-1 ROT R IDLE POS
AND       M04130	// R_1st ROT Y 1st POS
AND       T1804	// R-1st Cyl Clamp Up
AND       T1095	// R_4th DIE ALIGN BACKWARD
AND       T1096	// R_4th SIDE ALIGN BACKWARD
AND       P00065	// R_1st ROTATE MANDREL BACKWARD
MPUSH
AND       M12574	// R_1st MAND STEP 0
OUT       M12576	// R_1st MAND STEP INITIAL
MPOP
OUT       M12578	// R_1st MAND STEP INITIAL OK
// ======================== STEP ==========================
; L23
LOADP     M19046	// T)R_ALL STEP PLS
ORP       M12592	// T)R_1st MAND STEP+
OR        M12586	// R_1st MAND STEP KP
LOAD      M00211	// RT_AUTO RUN
OR        M12570	// R_1st MAND 1Cycle Run
AND LOAD
AND       M19044	// T)R_STEP MODE
AND NOT   T1060	// R_1st MAND STEP DELAY TM
AND NOT   M00105	// RIGHT STOP SW
AND NOT   M1259A	// R_1st MAND ORIGIN KP
AND NOT   T1063	// R_1st MAND CYCLE TIMEOUT
OUT       M12586	// R_1st MAND STEP KP
TON       T1063 5000	// R_1st MAND CYCLE TIMEOUT
// ======================== CYCLE RUN ==========================
; L27
LOAD NOT  T0055	// RT_AUTO RUN 1s
AND NOT   M12570	// R_1st MAND 1Cycle Run
NOT
LOAD      M12584	// R_1st MAND STEP ¾Æ´Ô
OR        M12586	// R_1st MAND STEP KP
AND LOAD
AND       F0009A
OUT       M12580	// R_1st MAND CYCLE RUN
; L29
LOAD      M12580	// R_1st MAND CYCLE RUN
AND       M12576	// R_1st MAND STEP INITIAL
OUT       M12582	// R_1st MAND CYCLE RUN PLS
; L30
LOADP     M12582	// R_1st MAND CYCLE RUN PLS
SET       M12510	// 06_On Vaccum
; L31
LOAD NOT  M19044	// T)R_STEP MODE
OUT       M12584	// R_1st MAND STEP ¾Æ´Ô

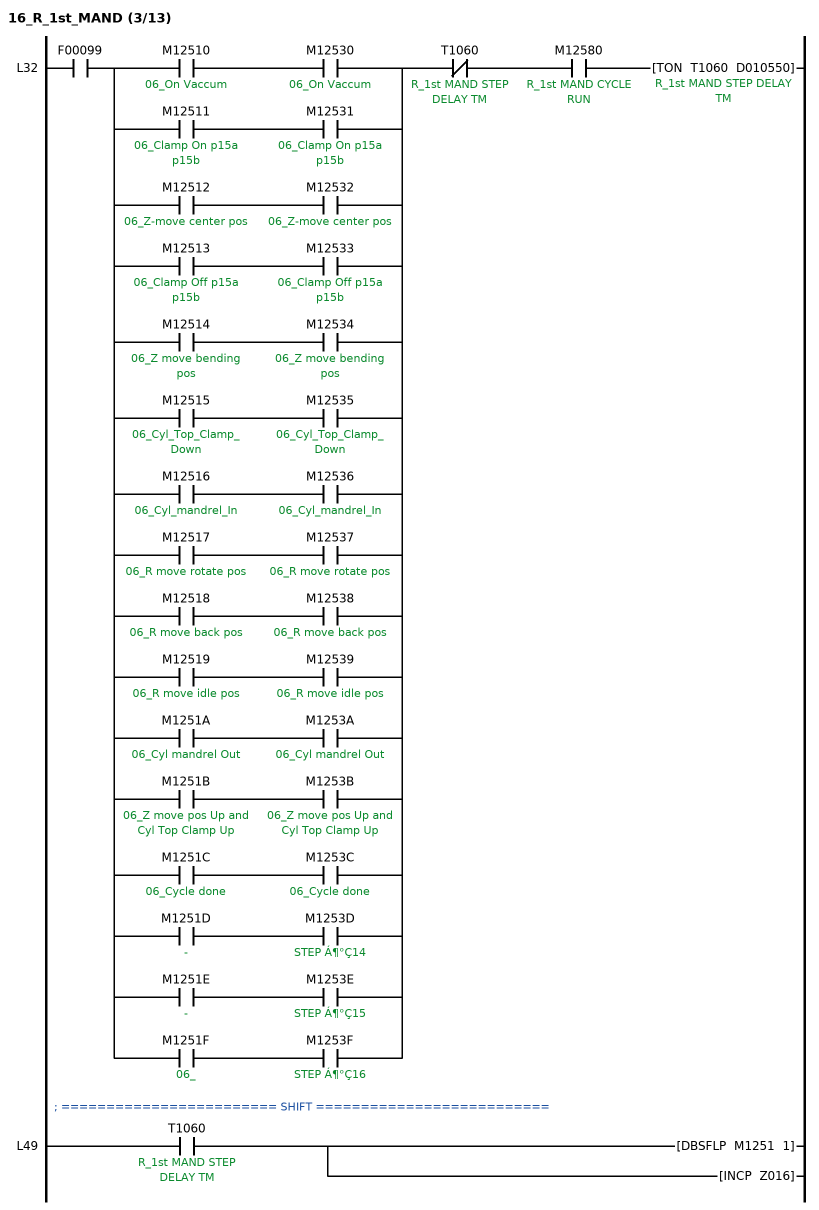
; L32
LOAD      F00099
LOAD      M12510	// 06_On Vaccum
AND       M12530	// 06_On Vaccum
LOAD      M12511	// 06_Clamp On p15a p15b
AND       M12531	// 06_Clamp On p15a p15b
OR LOAD
LOAD      M12512	// 06_Z-move center pos
AND       M12532	// 06_Z-move center pos
OR LOAD
LOAD      M12513	// 06_Clamp Off p15a p15b
AND       M12533	// 06_Clamp Off p15a p15b
OR LOAD
LOAD      M12514	// 06_Z move bending pos
AND       M12534	// 06_Z move bending pos
OR LOAD
LOAD      M12515	// 06_Cyl_Top_Clamp_Down
AND       M12535	// 06_Cyl_Top_Clamp_Down
OR LOAD
LOAD      M12516	// 06_Cyl_mandrel_In
AND       M12536	// 06_Cyl_mandrel_In
OR LOAD
LOAD      M12517	// 06_R move rotate pos
AND       M12537	// 06_R move rotate pos
OR LOAD
LOAD      M12518	// 06_R move back pos
AND       M12538	// 06_R move back pos
OR LOAD
LOAD      M12519	// 06_R move idle pos
AND       M12539	// 06_R move idle pos
OR LOAD
LOAD      M1251A	// 06_Cyl mandrel Out
AND       M1253A	// 06_Cyl mandrel Out
OR LOAD
LOAD      M1251B	// 06_Z move pos Up and Cyl Top Clamp Up
AND       M1253B	// 06_Z move pos Up and Cyl Top Clamp Up
OR LOAD
LOAD      M1251C	// 06_Cycle done
AND       M1253C	// 06_Cycle done
OR LOAD
LOAD      M1251D	// -
AND       M1253D	// STEP Á¶°Ç14
OR LOAD
LOAD      M1251E	// -
AND       M1253E	// STEP Á¶°Ç15
OR LOAD
LOAD      M1251F	// 06_
AND       M1253F	// STEP Á¶°Ç16
OR LOAD
AND LOAD
AND NOT   T1060	// R_1st MAND STEP DELAY TM
AND       M12580	// R_1st MAND CYCLE RUN
TON       T1060 D010550	// R_1st MAND STEP DELAY TM
// ======================== SHIFT ==========================
; L49
LOAD      T1060	// R_1st MAND STEP DELAY TM
DBSFLP    M1251 1
INCP      Z016

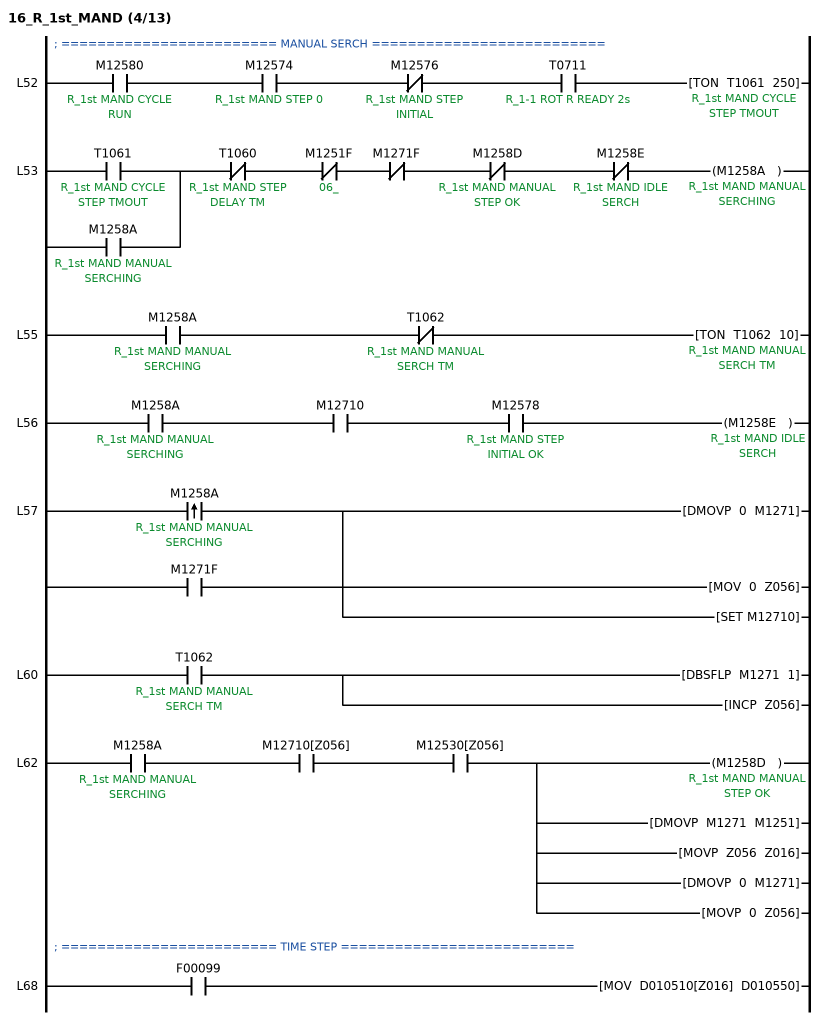
// ======================== MANUAL SERCH ==========================
; L52
LOAD      M12580	// R_1st MAND CYCLE RUN
AND       M12574	// R_1st MAND STEP 0
AND NOT   M12576	// R_1st MAND STEP INITIAL
AND       T0711	// R_1-1 ROT R READY 2s
TON       T1061 250	// R_1st MAND CYCLE STEP TMOUT
; L53
LOAD      T1061	// R_1st MAND CYCLE STEP TMOUT
OR        M1258A	// R_1st MAND MANUAL SERCHING
AND NOT   T1060	// R_1st MAND STEP DELAY TM
AND NOT   M1251F	// 06_
AND NOT   M1271F
AND NOT   M1258D	// R_1st MAND MANUAL STEP OK
AND NOT   M1258E	// R_1st MAND IDLE SERCH
OUT       M1258A	// R_1st MAND MANUAL SERCHING
; L55
LOAD      M1258A	// R_1st MAND MANUAL SERCHING
AND NOT   T1062	// R_1st MAND MANUAL SERCH TM
TON       T1062 10	// R_1st MAND MANUAL SERCH TM
; L56
LOAD      M1258A	// R_1st MAND MANUAL SERCHING
AND       M12710
AND       M12578	// R_1st MAND STEP INITIAL OK
OUT       M1258E	// R_1st MAND IDLE SERCH
; L57
LOADP     M1258A	// R_1st MAND MANUAL SERCHING
OR        M1271F
DMOVP     0 M1271
MOV       0 Z056
SET       M12710
; L60
LOAD      T1062	// R_1st MAND MANUAL SERCH TM
DBSFLP    M1271 1
INCP      Z056
; L62
LOAD      M1258A	// R_1st MAND MANUAL SERCHING
AND       M12710[Z056]
AND       M12530[Z056]
OUT       M1258D	// R_1st MAND MANUAL STEP OK
DMOVP     M1271 M1251
MOVP      Z056 Z016
DMOVP     0 M1271
MOVP      0 Z056
// ======================== TIME STEP ==========================
; L68
LOAD      F00099
MOV       D010510[Z016] D010550

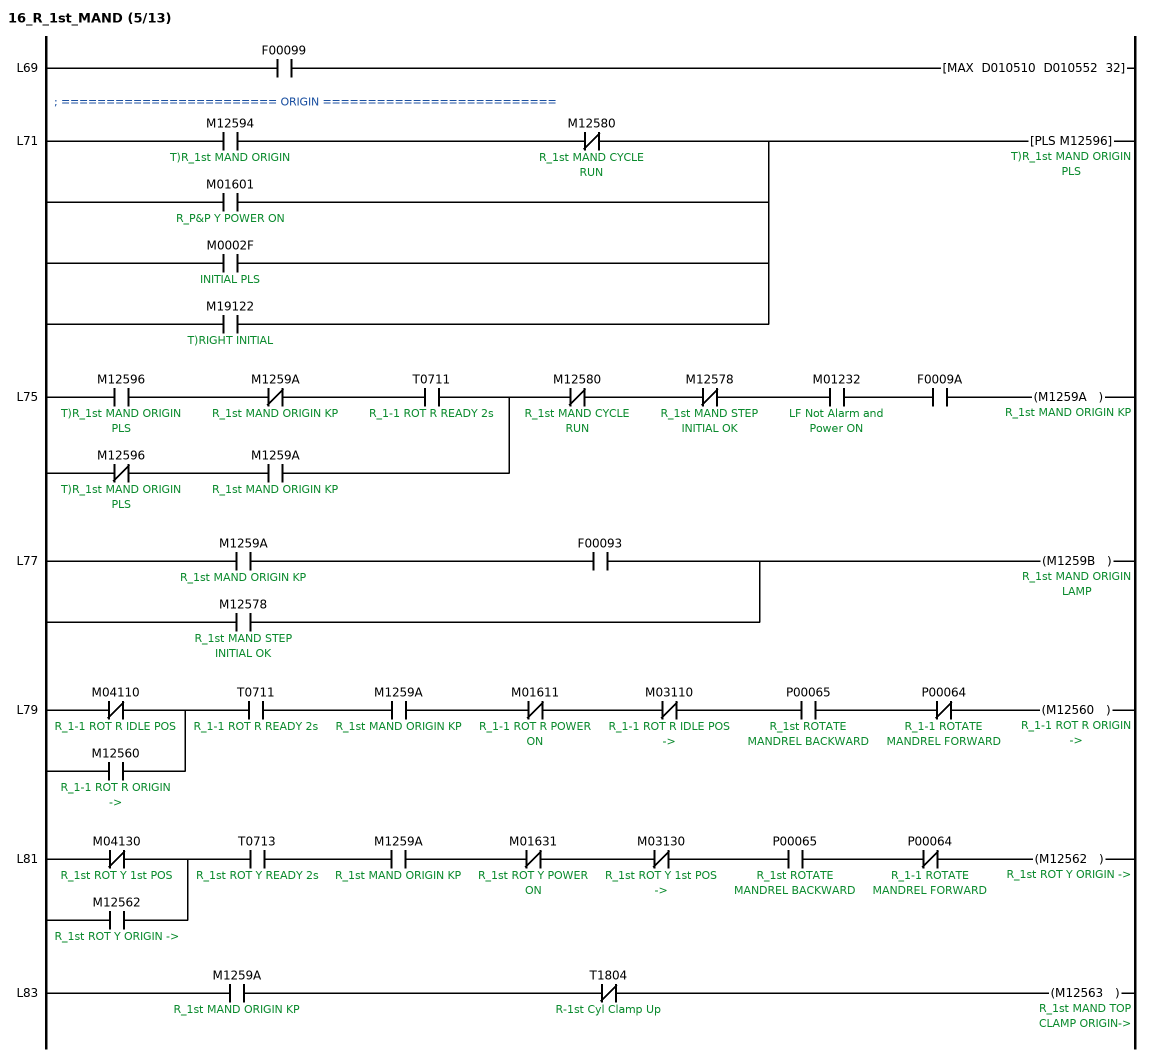
; L69
LOAD      F00099
MAX       D010510 D010552 32
// ======================== ORIGIN ==========================
; L71
LOAD      M12594	// T)R_1st MAND ORIGIN
AND NOT   M12580	// R_1st MAND CYCLE RUN
OR        M01601	// R_P&P Y POWER ON
OR        M0002F	// INITIAL PLS
OR        M19122	// T)RIGHT INITIAL
OUTP      M12596	// T)R_1st MAND ORIGIN PLS
; L75
LOAD      M12596	// T)R_1st MAND ORIGIN PLS
AND NOT   M1259A	// R_1st MAND ORIGIN KP
AND       T0711	// R_1-1 ROT R READY 2s
LOAD NOT  M12596	// T)R_1st MAND ORIGIN PLS
AND       M1259A	// R_1st MAND ORIGIN KP
OR LOAD
AND NOT   M12580	// R_1st MAND CYCLE RUN
AND NOT   M12578	// R_1st MAND STEP INITIAL OK
AND       M01232	// LF Not Alarm and Power ON
AND       F0009A
OUT       M1259A	// R_1st MAND ORIGIN KP
; L77
LOAD      M1259A	// R_1st MAND ORIGIN KP
AND       F00093
OR        M12578	// R_1st MAND STEP INITIAL OK
OUT       M1259B	// R_1st MAND ORIGIN LAMP
; L79
LOAD NOT  M04110	// R_1-1 ROT R IDLE POS
OR        M12560	// R_1-1 ROT R ORIGIN ->
AND       T0711	// R_1-1 ROT R READY 2s
AND       M1259A	// R_1st MAND ORIGIN KP
AND NOT   M01611	// R_1-1 ROT R POWER ON
AND NOT   M03110	// R_1-1 ROT R IDLE POS ->
AND       P00065	// R_1st ROTATE MANDREL BACKWARD
AND NOT   P00064	// R_1-1 ROTATE MANDREL FORWARD
OUT       M12560	// R_1-1 ROT R ORIGIN ->
; L81
LOAD NOT  M04130	// R_1st ROT Y 1st POS
OR        M12562	// R_1st ROT Y ORIGIN ->
AND       T0713	// R_1st ROT Y READY 2s
AND       M1259A	// R_1st MAND ORIGIN KP
AND NOT   M01631	// R_1st ROT Y POWER ON
AND NOT   M03130	// R_1st ROT Y 1st POS ->
AND       P00065	// R_1st ROTATE MANDREL BACKWARD
AND NOT   P00064	// R_1-1 ROTATE MANDREL FORWARD
OUT       M12562	// R_1st ROT Y ORIGIN ->
; L83
LOAD      M1259A	// R_1st MAND ORIGIN KP
AND NOT   T1804	// R-1st Cyl Clamp Up
OUT       M12563	// R_1st MAND TOP CLAMP ORIGIN->

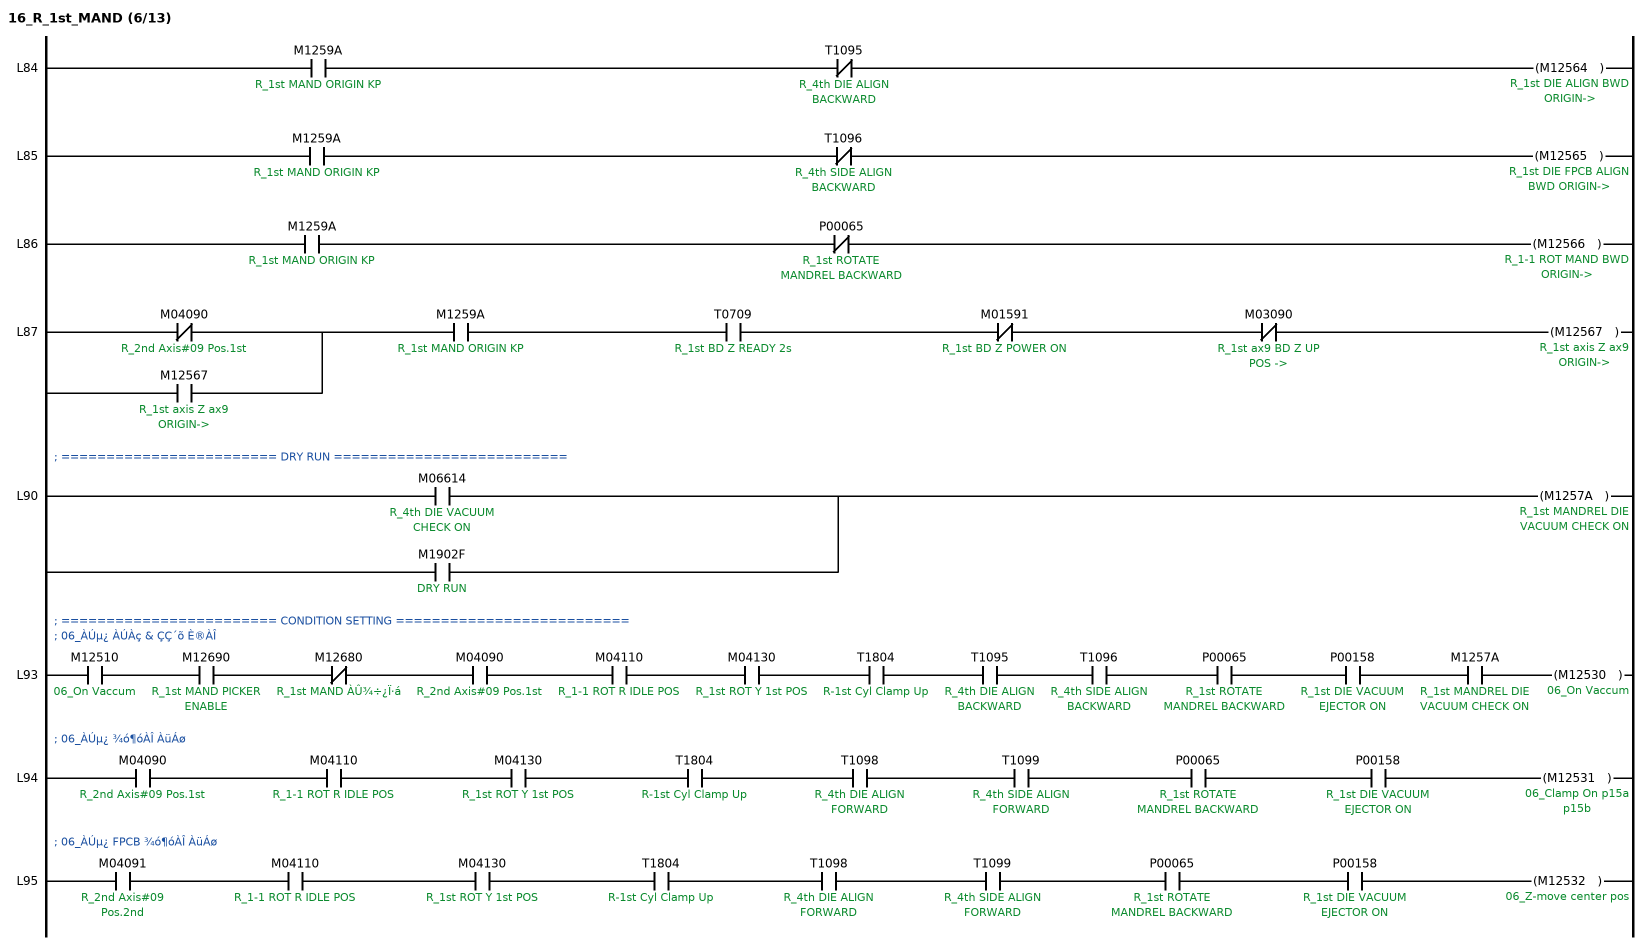
; L84
LOAD      M1259A	// R_1st MAND ORIGIN KP
AND NOT   T1095	// R_4th DIE ALIGN BACKWARD
OUT       M12564	// R_1st DIE ALIGN BWD ORIGIN->
; L85
LOAD      M1259A	// R_1st MAND ORIGIN KP
AND NOT   T1096	// R_4th SIDE ALIGN BACKWARD
OUT       M12565	// R_1st DIE FPCB ALIGN BWD ORIGIN->
; L86
LOAD      M1259A	// R_1st MAND ORIGIN KP
AND NOT   P00065	// R_1st ROTATE MANDREL BACKWARD
OUT       M12566	// R_1-1 ROT MAND BWD ORIGIN->
; L87
LOAD NOT  M04090	// R_2nd Axis#09 Pos.1st
OR        M12567	// R_1st axis Z ax9 ORIGIN->
AND       M1259A	// R_1st MAND ORIGIN KP
AND       T0709	// R_1st BD Z READY 2s
AND NOT   M01591	// R_1st BD Z POWER ON
AND NOT   M03090	// R_1st ax9 BD Z UP POS ->
OUT       M12567	// R_1st axis Z ax9 ORIGIN->
// ======================== DRY RUN ==========================
; L90
LOAD      M06614	// R_4th DIE VACUUM CHECK ON
OR        M1902F	// DRY RUN
OUT       M1257A	// R_1st MANDREL DIE VACUUM CHECK ON
// ======================== CONDITION SETTING ==========================
; L93
LOAD      M12510	// 06_On Vaccum
AND       M12690	// R_1st MAND PICKER ENABLE
AND NOT   M12680	// R_1st MAND ÀÛ¾÷¿Ï·á
AND       M04090	// R_2nd Axis#09 Pos.1st
AND       M04110	// R_1-1 ROT R IDLE POS
AND       M04130	// R_1st ROT Y 1st POS
AND       T1804	// R-1st Cyl Clamp Up
AND       T1095	// R_4th DIE ALIGN BACKWARD
AND       T1096	// R_4th SIDE ALIGN BACKWARD
AND       P00065	// R_1st ROTATE MANDREL BACKWARD
AND       P00158	// R_1st DIE VACUUM EJECTOR ON
AND       M1257A	// R_1st MANDREL DIE VACUUM CHECK ON
OUT       M12530	// 06_On Vaccum
// output comment: 06_ÀÚµ¿ ÀÚÀç & ÇÇ´õ È®ÀÎ
; L94
LOAD      M04090	// R_2nd Axis#09 Pos.1st
AND       M04110	// R_1-1 ROT R IDLE POS
AND       M04130	// R_1st ROT Y 1st POS
AND       T1804	// R-1st Cyl Clamp Up
AND       T1098	// R_4th DIE ALIGN FORWARD
AND       T1099	// R_4th SIDE ALIGN FORWARD
AND       P00065	// R_1st ROTATE MANDREL BACKWARD
AND       P00158	// R_1st DIE VACUUM EJECTOR ON
OUT       M12531	// 06_Clamp On p15a p15b
// output comment: 06_ÀÚµ¿ ¾ó¶óÀÎ ÀüÁø
; L95
LOAD      M04091	// R_2nd Axis#09 Pos.2nd
AND       M04110	// R_1-1 ROT R IDLE POS
AND       M04130	// R_1st ROT Y 1st POS
AND       T1804	// R-1st Cyl Clamp Up
AND       T1098	// R_4th DIE ALIGN FORWARD
AND       T1099	// R_4th SIDE ALIGN FORWARD
AND       P00065	// R_1st ROTATE MANDREL BACKWARD
AND       P00158	// R_1st DIE VACUUM EJECTOR ON
OUT       M12532	// 06_Z-move center pos
// output comment: 06_ÀÚµ¿ FPCB ¾ó¶óÀÎ ÀüÁø

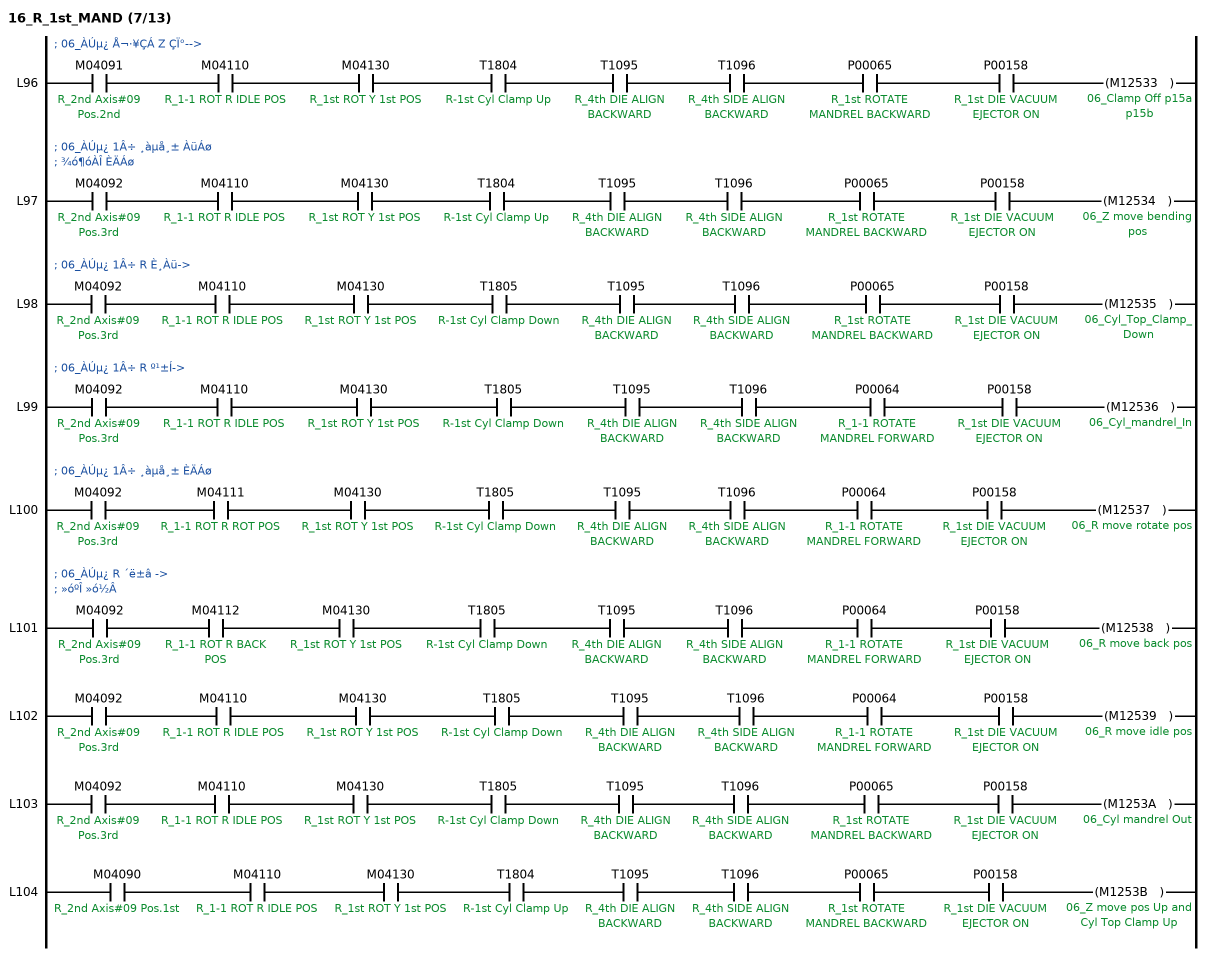
; L96
LOAD      M04091	// R_2nd Axis#09 Pos.2nd
AND       M04110	// R_1-1 ROT R IDLE POS
AND       M04130	// R_1st ROT Y 1st POS
AND       T1804	// R-1st Cyl Clamp Up
AND       T1095	// R_4th DIE ALIGN BACKWARD
AND       T1096	// R_4th SIDE ALIGN BACKWARD
AND       P00065	// R_1st ROTATE MANDREL BACKWARD
AND       P00158	// R_1st DIE VACUUM EJECTOR ON
OUT       M12533	// 06_Clamp Off p15a p15b
// output comment: 06_ÀÚµ¿ Å¬·¥ÇÁ Z ÇÏ°­->
; L97
LOAD      M04092	// R_2nd Axis#09 Pos.3rd
AND       M04110	// R_1-1 ROT R IDLE POS
AND       M04130	// R_1st ROT Y 1st POS
AND       T1804	// R-1st Cyl Clamp Up
AND       T1095	// R_4th DIE ALIGN BACKWARD
AND       T1096	// R_4th SIDE ALIGN BACKWARD
AND       P00065	// R_1st ROTATE MANDREL BACKWARD
AND       P00158	// R_1st DIE VACUUM EJECTOR ON
OUT       M12534	// 06_Z move bending pos
// output comment: 06_ÀÚµ¿ 1Â÷ ¸àµå¸± ÀüÁø ¾ó¶óÀÎ ÈÄÁø
; L98
LOAD      M04092	// R_2nd Axis#09 Pos.3rd
AND       M04110	// R_1-1 ROT R IDLE POS
AND       M04130	// R_1st ROT Y 1st POS
AND       T1805	// R-1st Cyl Clamp Down
AND       T1095	// R_4th DIE ALIGN BACKWARD
AND       T1096	// R_4th SIDE ALIGN BACKWARD
AND       P00065	// R_1st ROTATE MANDREL BACKWARD
AND       P00158	// R_1st DIE VACUUM EJECTOR ON
OUT       M12535	// 06_Cyl_Top_Clamp_Down
// output comment: 06_ÀÚµ¿ 1Â÷ R È¸Àü->
; L99
LOAD      M04092	// R_2nd Axis#09 Pos.3rd
AND       M04110	// R_1-1 ROT R IDLE POS
AND       M04130	// R_1st ROT Y 1st POS
AND       T1805	// R-1st Cyl Clamp Down
AND       T1095	// R_4th DIE ALIGN BACKWARD
AND       T1096	// R_4th SIDE ALIGN BACKWARD
AND       P00064	// R_1-1 ROTATE MANDREL FORWARD
AND       P00158	// R_1st DIE VACUUM EJECTOR ON
OUT       M12536	// 06_Cyl_mandrel_In
// output comment: 06_ÀÚµ¿ 1Â÷ R º¹±Í->
; L100
LOAD      M04092	// R_2nd Axis#09 Pos.3rd
AND       M04111	// R_1-1 ROT R ROT POS
AND       M04130	// R_1st ROT Y 1st POS
AND       T1805	// R-1st Cyl Clamp Down
AND       T1095	// R_4th DIE ALIGN BACKWARD
AND       T1096	// R_4th SIDE ALIGN BACKWARD
AND       P00064	// R_1-1 ROTATE MANDREL FORWARD
AND       P00158	// R_1st DIE VACUUM EJECTOR ON
OUT       M12537	// 06_R move rotate pos
// output comment: 06_ÀÚµ¿ 1Â÷ ¸àµå¸± ÈÄÁø
; L101
LOAD      M04092	// R_2nd Axis#09 Pos.3rd
AND       M04112	// R_1-1 ROT R BACK POS
AND       M04130	// R_1st ROT Y 1st POS
AND       T1805	// R-1st Cyl Clamp Down
AND       T1095	// R_4th DIE ALIGN BACKWARD
AND       T1096	// R_4th SIDE ALIGN BACKWARD
AND       P00064	// R_1-1 ROTATE MANDREL FORWARD
AND       P00158	// R_1st DIE VACUUM EJECTOR ON
OUT       M12538	// 06_R move back pos
// output comment: 06_ÀÚµ¿ R ´ë±â -> »óºÎ »ó½Â
; L102
LOAD      M04092	// R_2nd Axis#09 Pos.3rd
AND       M04110	// R_1-1 ROT R IDLE POS
AND       M04130	// R_1st ROT Y 1st POS
AND       T1805	// R-1st Cyl Clamp Down
AND       T1095	// R_4th DIE ALIGN BACKWARD
AND       T1096	// R_4th SIDE ALIGN BACKWARD
AND       P00064	// R_1-1 ROTATE MANDREL FORWARD
AND       P00158	// R_1st DIE VACUUM EJECTOR ON
OUT       M12539	// 06_R move idle pos
; L103
LOAD      M04092	// R_2nd Axis#09 Pos.3rd
AND       M04110	// R_1-1 ROT R IDLE POS
AND       M04130	// R_1st ROT Y 1st POS
AND       T1805	// R-1st Cyl Clamp Down
AND       T1095	// R_4th DIE ALIGN BACKWARD
AND       T1096	// R_4th SIDE ALIGN BACKWARD
AND       P00065	// R_1st ROTATE MANDREL BACKWARD
AND       P00158	// R_1st DIE VACUUM EJECTOR ON
OUT       M1253A	// 06_Cyl mandrel Out
; L104
LOAD      M04090	// R_2nd Axis#09 Pos.1st
AND       M04110	// R_1-1 ROT R IDLE POS
AND       M04130	// R_1st ROT Y 1st POS
AND       T1804	// R-1st Cyl Clamp Up
AND       T1095	// R_4th DIE ALIGN BACKWARD
AND       T1096	// R_4th SIDE ALIGN BACKWARD
AND       P00065	// R_1st ROTATE MANDREL BACKWARD
AND       P00158	// R_1st DIE VACUUM EJECTOR ON
OUT       M1253B	// 06_Z move pos Up and Cyl Top Clamp Up

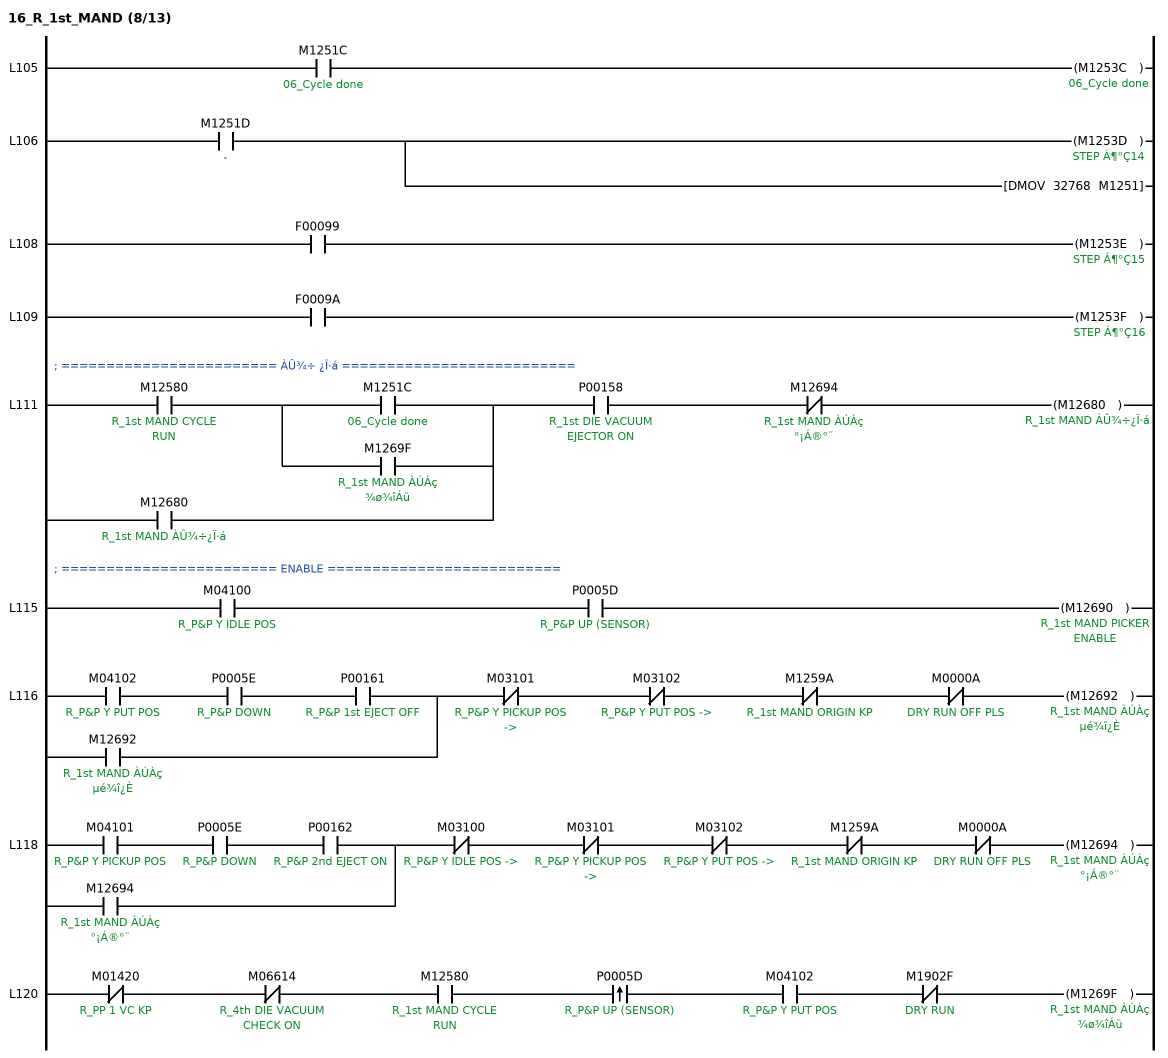
; L105
LOAD      M1251C	// 06_Cycle done
OUT       M1253C	// 06_Cycle done
; L106
LOAD      M1251D	// -
OUT       M1253D	// STEP Á¶°Ç14
DMOV      32768 M1251
; L108
LOAD      F00099
OUT       M1253E	// STEP Á¶°Ç15
; L109
LOAD      F0009A
OUT       M1253F	// STEP Á¶°Ç16
// ======================== ÀÛ¾÷ ¿Ï·á ==========================
; L111
LOAD      M12580	// R_1st MAND CYCLE RUN
LOAD      M1251C	// 06_Cycle done
OR        M1269F	// R_1st MAND ÀÚÀç ¾ø¾îÁü
AND LOAD
OR        M12680	// R_1st MAND ÀÛ¾÷¿Ï·á
AND       P00158	// R_1st DIE VACUUM EJECTOR ON
AND NOT   M12694	// R_1st MAND ÀÚÀç °¡Á®°¨
OUT       M12680	// R_1st MAND ÀÛ¾÷¿Ï·á
// ======================== ENABLE ==========================
; L115
LOAD      M04100	// R_P&P Y IDLE POS
AND       P0005D	// R_P&P UP (SENSOR)
OUT       M12690	// R_1st MAND PICKER ENABLE
; L116
LOAD      M04102	// R_P&P Y PUT POS
AND       P0005E	// R_P&P DOWN
AND       P00161	// R_P&P 1st EJECT OFF
OR        M12692	// R_1st MAND ÀÚÀç µé¾î¿È
AND NOT   M03101	// R_P&P Y PICKUP POS ->
AND NOT   M03102	// R_P&P Y PUT POS ->
AND NOT   M1259A	// R_1st MAND ORIGIN KP
AND NOT   M0000A	// DRY RUN OFF PLS
OUT       M12692	// R_1st MAND ÀÚÀç µé¾î¿È
; L118
LOAD      M04101	// R_P&P Y PICKUP POS
AND       P0005E	// R_P&P DOWN
AND       P00162	// R_P&P 2nd EJECT ON
OR        M12694	// R_1st MAND ÀÚÀç °¡Á®°¨
AND NOT   M03100	// R_P&P Y IDLE POS ->
AND NOT   M03101	// R_P&P Y PICKUP POS ->
AND NOT   M03102	// R_P&P Y PUT POS ->
AND NOT   M1259A	// R_1st MAND ORIGIN KP
AND NOT   M0000A	// DRY RUN OFF PLS
OUT       M12694	// R_1st MAND ÀÚÀç °¡Á®°¨
; L120
LOAD NOT  M01420	// R_PP 1 VC KP
AND NOT   M06614	// R_4th DIE VACUUM CHECK ON
AND       M12580	// R_1st MAND CYCLE RUN
ANDP      P0005D	// R_P&P UP (SENSOR)
AND       M04102	// R_P&P Y PUT POS
AND NOT   M1902F	// DRY RUN
OUT       M1269F	// R_1st MAND ÀÚÀç ¾ø¾îÁü

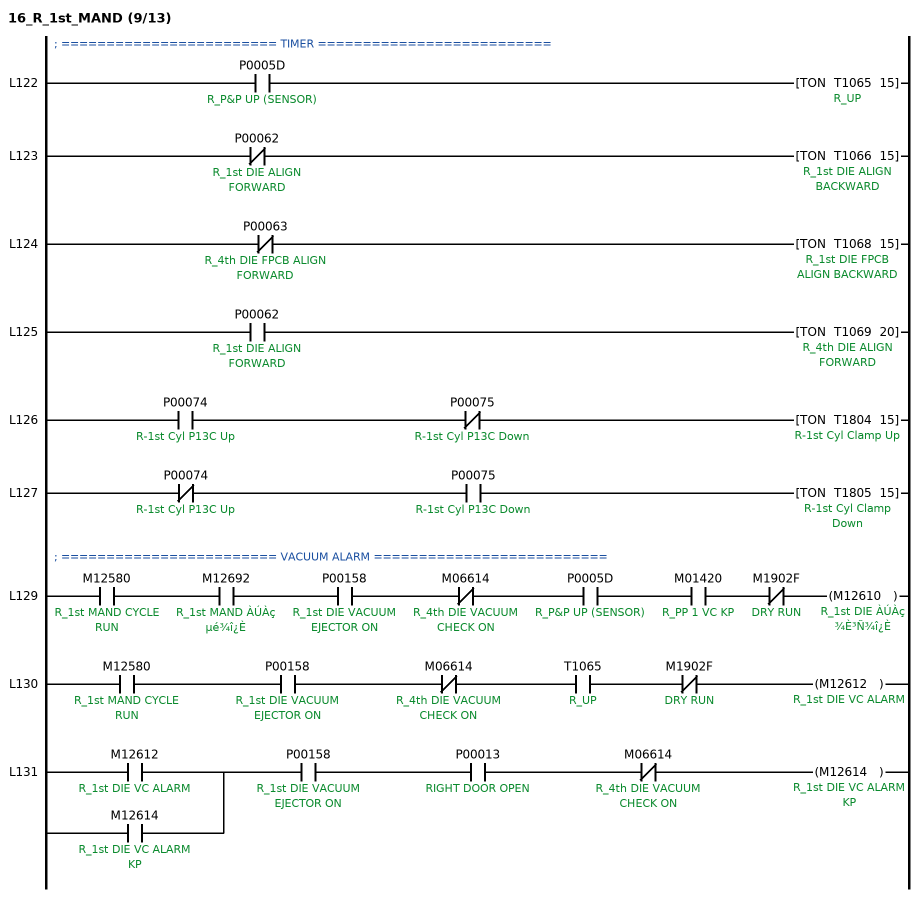
// ======================== TIMER ==========================
; L122
LOAD      P0005D	// R_P&P UP (SENSOR)
TON       T1065 15	// R_UP
; L123
LOAD NOT  P00062	// R_1st DIE ALIGN FORWARD
TON       T1066 15	// R_1st DIE ALIGN BACKWARD
; L124
LOAD NOT  P00063	// R_4th DIE FPCB ALIGN FORWARD
TON       T1068 15	// R_1st DIE FPCB ALIGN BACKWARD
; L125
LOAD      P00062	// R_1st DIE ALIGN FORWARD
TON       T1069 20	// R_4th DIE ALIGN FORWARD
; L126
LOAD      P00074	// R-1st Cyl P13C Up
AND NOT   P00075	// R-1st Cyl P13C Down
TON       T1804 15	// R-1st Cyl Clamp Up
; L127
LOAD NOT  P00074	// R-1st Cyl P13C Up
AND       P00075	// R-1st Cyl P13C Down
TON       T1805 15	// R-1st Cyl Clamp Down
// ======================== VACUUM ALARM ==========================
; L129
LOAD      M12580	// R_1st MAND CYCLE RUN
AND       M12692	// R_1st MAND ÀÚÀç µé¾î¿È
AND       P00158	// R_1st DIE VACUUM EJECTOR ON
AND NOT   M06614	// R_4th DIE VACUUM CHECK ON
AND       P0005D	// R_P&P UP (SENSOR)
AND       M01420	// R_PP 1 VC KP
AND NOT   M1902F	// DRY RUN
OUT       M12610	// R_1st DIE ÀÚÀç ¾È³Ñ¾î¿È
; L130
LOAD      M12580	// R_1st MAND CYCLE RUN
AND       P00158	// R_1st DIE VACUUM EJECTOR ON
AND NOT   M06614	// R_4th DIE VACUUM CHECK ON
AND       T1065	// R_UP
AND NOT   M1902F	// DRY RUN
OUT       M12612	// R_1st DIE VC ALARM
; L131
LOAD      M12612	// R_1st DIE VC ALARM
OR        M12614	// R_1st DIE VC ALARM KP
AND       P00158	// R_1st DIE VACUUM EJECTOR ON
AND       P00013	// RIGHT DOOR OPEN
AND NOT   M06614	// R_4th DIE VACUUM CHECK ON
OUT       M12614	// R_1st DIE VC ALARM KP

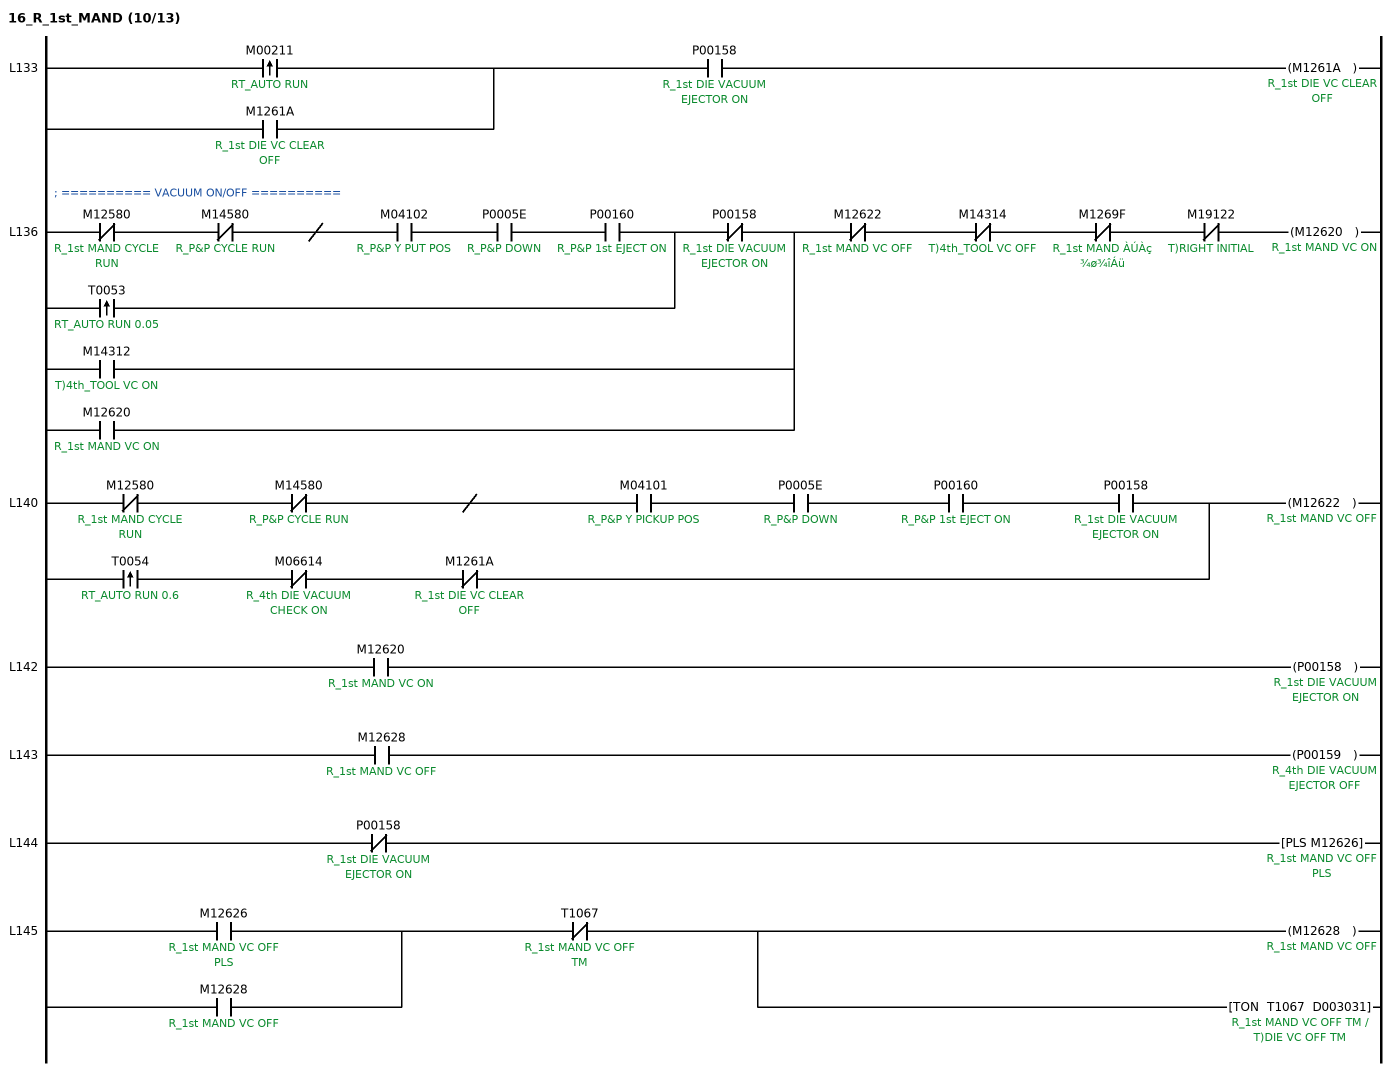
; L133
LOADP     M00211	// RT_AUTO RUN
OR        M1261A	// R_1st DIE VC CLEAR OFF
AND       P00158	// R_1st DIE VACUUM EJECTOR ON
OUT       M1261A	// R_1st DIE VC CLEAR OFF
// ========== VACUUM ON/OFF ==========
; L136
LOAD NOT  M12580	// R_1st MAND CYCLE RUN
AND NOT   M14580	// R_P&P CYCLE RUN
NOT
AND       M04102	// R_P&P Y PUT POS
AND       P0005E	// R_P&P DOWN
AND       P00160	// R_P&P 1st EJECT ON
ORP       T0053	// RT_AUTO RUN 0.05
AND NOT   P00158	// R_1st DIE VACUUM EJECTOR ON
OR        M14312	// T)4th_TOOL VC ON
OR        M12620	// R_1st MAND VC ON
AND NOT   M12622	// R_1st MAND VC OFF
AND NOT   M14314	// T)4th_TOOL VC OFF
AND NOT   M1269F	// R_1st MAND ÀÚÀç ¾ø¾îÁü
AND NOT   M19122	// T)RIGHT INITIAL
OUT       M12620	// R_1st MAND VC ON
; L140
LOAD NOT  M12580	// R_1st MAND CYCLE RUN
AND NOT   M14580	// R_P&P CYCLE RUN
NOT
AND       M04101	// R_P&P Y PICKUP POS
AND       P0005E	// R_P&P DOWN
AND       P00160	// R_P&P 1st EJECT ON
AND       P00158	// R_1st DIE VACUUM EJECTOR ON
LOADP     T0054	// RT_AUTO RUN 0.6
AND NOT   M06614	// R_4th DIE VACUUM CHECK ON
AND NOT   M1261A	// R_1st DIE VC CLEAR OFF
OR LOAD
OUT       M12622	// R_1st MAND VC OFF
; L142
LOAD      M12620	// R_1st MAND VC ON
OUT       P00158	// R_1st DIE VACUUM EJECTOR ON
; L143
LOAD      M12628	// R_1st MAND VC OFF
OUT       P00159	// R_4th DIE VACUUM EJECTOR OFF
; L144
LOAD NOT  P00158	// R_1st DIE VACUUM EJECTOR ON
OUTP      M12626	// R_1st MAND VC OFF PLS
; L145
LOAD      M12626	// R_1st MAND VC OFF PLS
OR        M12628	// R_1st MAND VC OFF
AND NOT   T1067	// R_1st MAND VC OFF TM
OUT       M12628	// R_1st MAND VC OFF
TON       T1067 D003031	// R_1st MAND VC OFF TM / T)DIE VC OFF TM

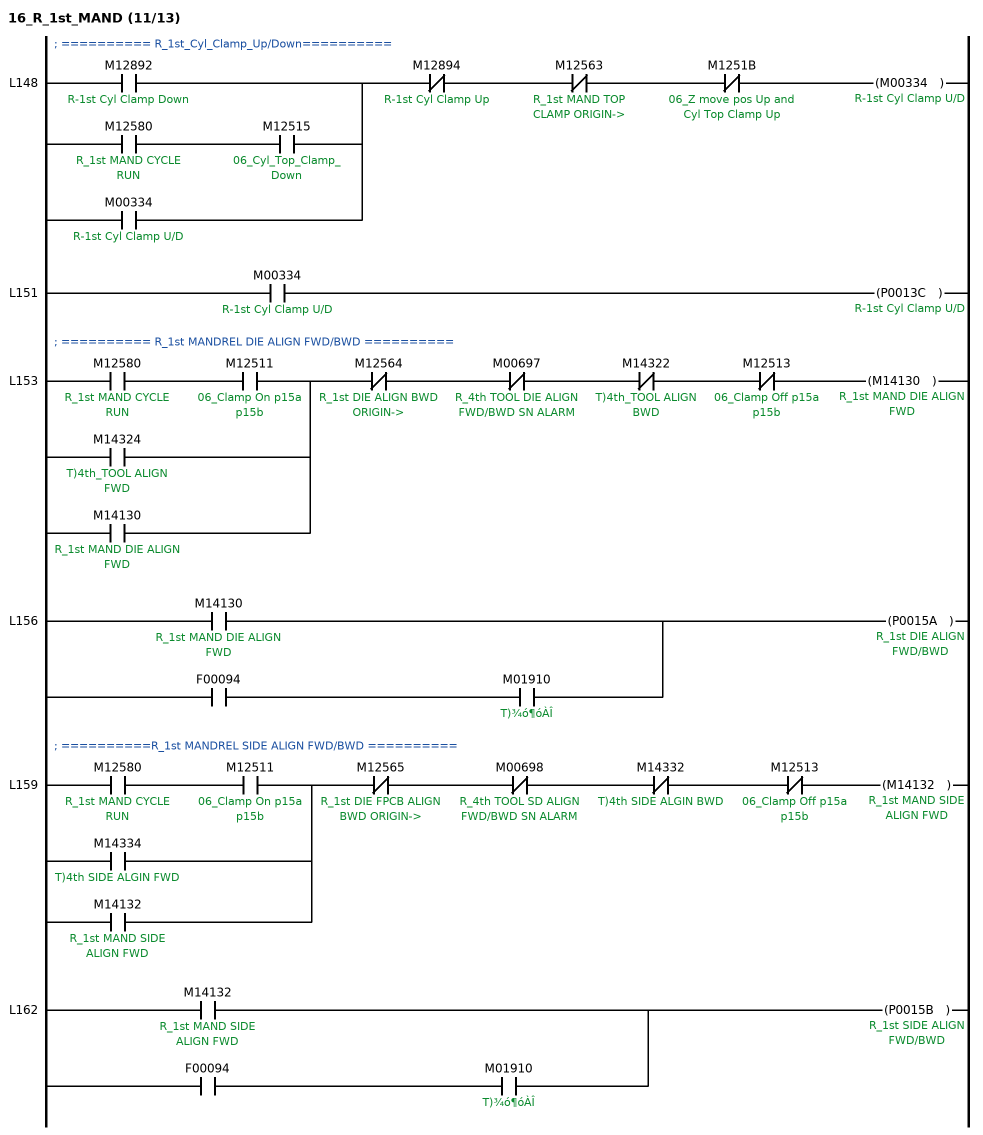
// ========== R_1st_Cyl_Clamp_Up/Down==========
; L148
LOAD      M12892	// R-1st Cyl Clamp Down
LOAD      M12580	// R_1st MAND CYCLE RUN
AND       M12515	// 06_Cyl_Top_Clamp_Down
OR LOAD
OR        M00334	// R-1st Cyl Clamp U/D
AND NOT   M12894	// R-1st Cyl Clamp Up
AND NOT   M12563	// R_1st MAND TOP CLAMP ORIGIN->
AND NOT   M1251B	// 06_Z move pos Up and Cyl Top Clamp Up
OUT       M00334	// R-1st Cyl Clamp U/D
; L151
LOAD      M00334	// R-1st Cyl Clamp U/D
OUT       P0013C	// R-1st Cyl Clamp U/D
// ========== R_1st MANDREL DIE ALIGN FWD/BWD ==========
; L153
LOAD      M12580	// R_1st MAND CYCLE RUN
AND       M12511	// 06_Clamp On p15a p15b
OR        M14324	// T)4th_TOOL ALIGN FWD
OR        M14130	// R_1st MAND DIE ALIGN FWD
AND NOT   M12564	// R_1st DIE ALIGN BWD ORIGIN->
AND NOT   M00697	// R_4th TOOL DIE ALIGN FWD/BWD SN ALARM
AND NOT   M14322	// T)4th_TOOL ALIGN BWD
AND NOT   M12513	// 06_Clamp Off p15a p15b
OUT       M14130	// R_1st MAND DIE ALIGN FWD
; L156
LOAD      M14130	// R_1st MAND DIE ALIGN FWD
LOAD      F00094
AND       M01910	// T)¾ó¶óÀÎ
OR LOAD
OUT       P0015A	// R_1st DIE ALIGN FWD/BWD
// ==========R_1st MANDREL SIDE ALIGN FWD/BWD ==========
; L159
LOAD      M12580	// R_1st MAND CYCLE RUN
AND       M12511	// 06_Clamp On p15a p15b
OR        M14334	// T)4th SIDE ALGIN FWD
OR        M14132	// R_1st MAND SIDE ALIGN FWD
AND NOT   M12565	// R_1st DIE FPCB ALIGN BWD ORIGIN->
AND NOT   M00698	// R_4th TOOL SD ALIGN FWD/BWD SN ALARM
AND NOT   M14332	// T)4th SIDE ALGIN BWD
AND NOT   M12513	// 06_Clamp Off p15a p15b
OUT       M14132	// R_1st MAND SIDE ALIGN FWD
; L162
LOAD      M14132	// R_1st MAND SIDE ALIGN FWD
LOAD      F00094
AND       M01910	// T)¾ó¶óÀÎ
OR LOAD
OUT       P0015B	// R_1st SIDE ALIGN FWD/BWD

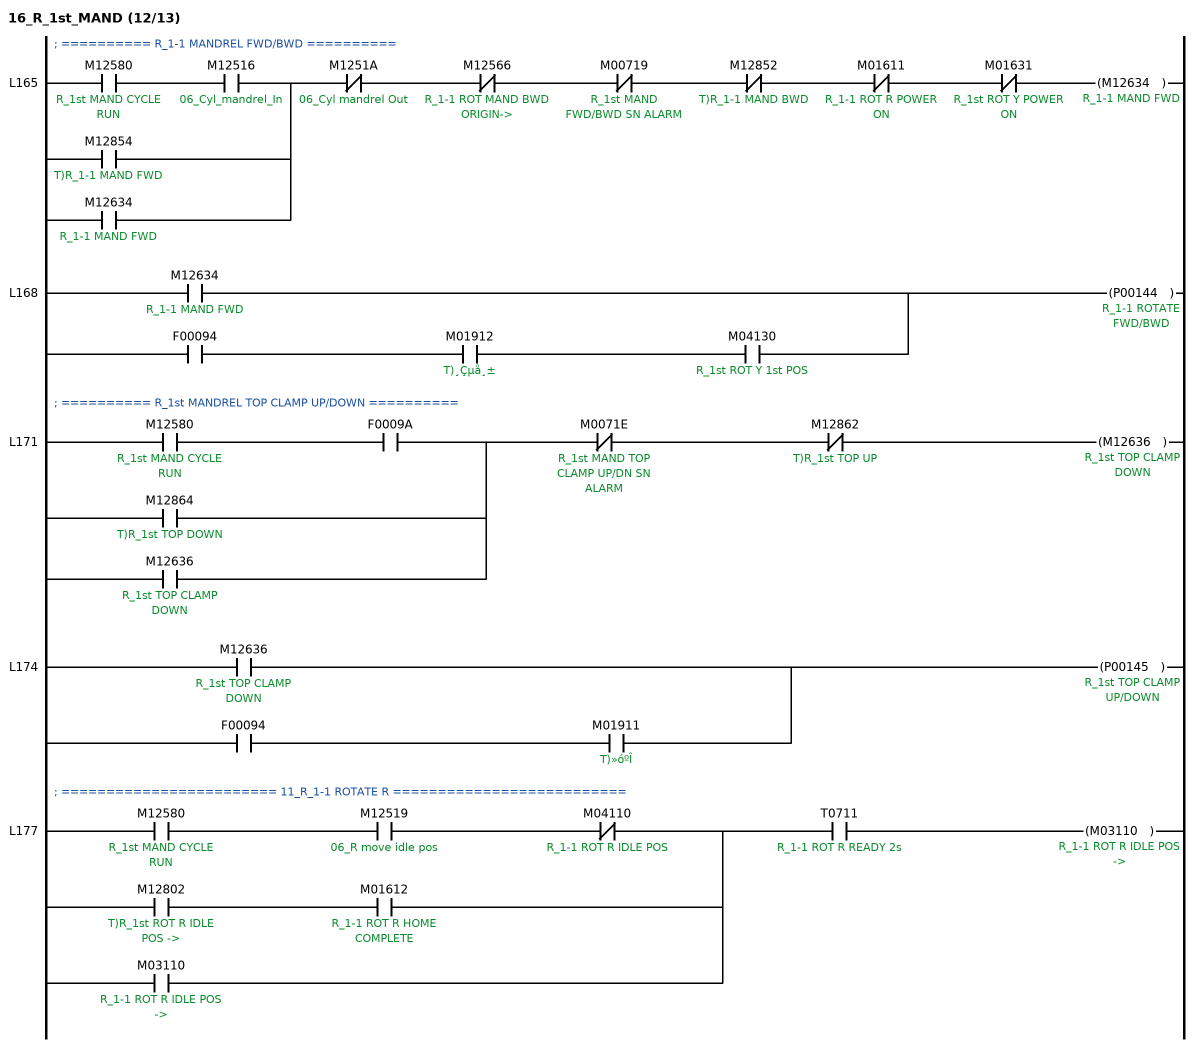
// ========== R_1-1 MANDREL FWD/BWD ==========
; L165
LOAD      M12580	// R_1st MAND CYCLE RUN
AND       M12516	// 06_Cyl_mandrel_In
OR        M12854	// T)R_1-1 MAND FWD
OR        M12634	// R_1-1 MAND FWD
AND NOT   M1251A	// 06_Cyl mandrel Out
AND NOT   M12566	// R_1-1 ROT MAND BWD ORIGIN->
AND NOT   M00719	// R_1st MAND FWD/BWD SN ALARM
AND NOT   M12852	// T)R_1-1 MAND BWD
AND NOT   M01611	// R_1-1 ROT R POWER ON
AND NOT   M01631	// R_1st ROT Y POWER ON
OUT       M12634	// R_1-1 MAND FWD
; L168
LOAD      M12634	// R_1-1 MAND FWD
LOAD      F00094
AND       M01912	// T)¸Çµå¸±
AND       M04130	// R_1st ROT Y 1st POS
OR LOAD
OUT       P00144	// R_1-1 ROTATE FWD/BWD
// ========== R_1st MANDREL TOP CLAMP UP/DOWN ==========
; L171
LOAD      M12580	// R_1st MAND CYCLE RUN
AND       F0009A
OR        M12864	// T)R_1st TOP DOWN
OR        M12636	// R_1st TOP CLAMP DOWN
AND NOT   M0071E	// R_1st MAND TOP CLAMP UP/DN SN ALARM
AND NOT   M12862	// T)R_1st TOP UP
OUT       M12636	// R_1st TOP CLAMP DOWN
; L174
LOAD      M12636	// R_1st TOP CLAMP DOWN
LOAD      F00094
AND       M01911	// T)»óºÎ
OR LOAD
OUT       P00145	// R_1st TOP CLAMP UP/DOWN
// ======================== 11_R_1-1 ROTATE R ==========================
; L177
LOAD      M12580	// R_1st MAND CYCLE RUN
AND       M12519	// 06_R move idle pos
AND NOT   M04110	// R_1-1 ROT R IDLE POS
LOAD      M12802	// T)R_1st ROT R IDLE POS ->
AND       M01612	// R_1-1 ROT R HOME COMPLETE
OR LOAD
OR        M03110	// R_1-1 ROT R IDLE POS ->
AND       T0711	// R_1-1 ROT R READY 2s
OUT       M03110	// R_1-1 ROT R IDLE POS ->

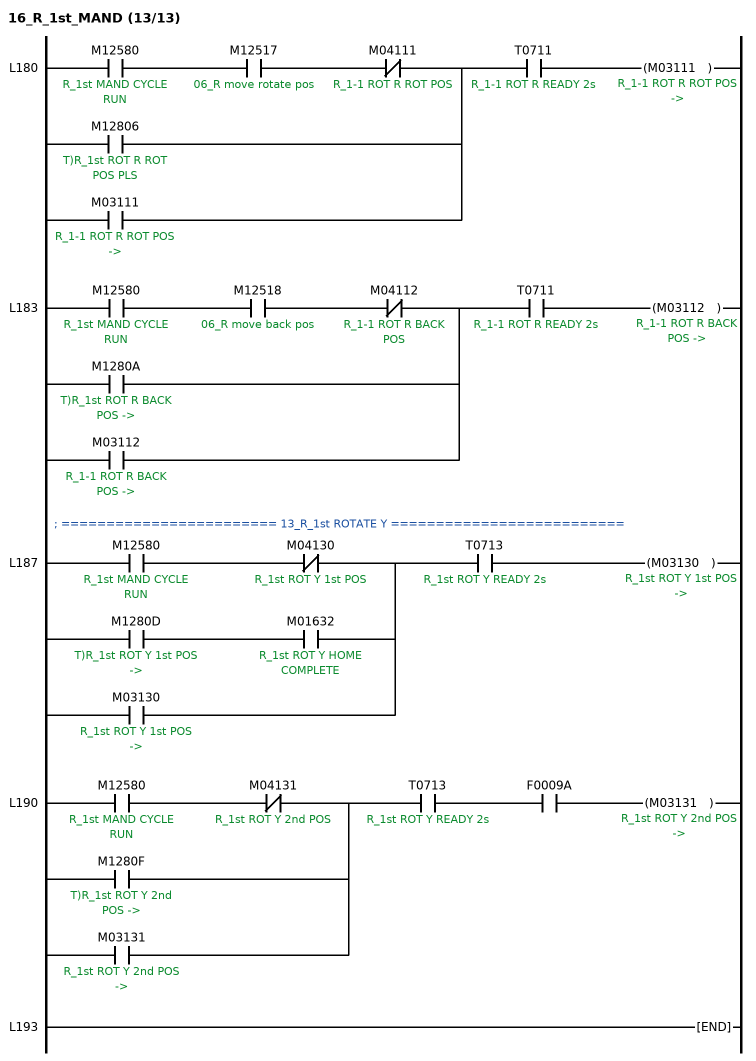
; L180
LOAD      M12580	// R_1st MAND CYCLE RUN
AND       M12517	// 06_R move rotate pos
AND NOT   M04111	// R_1-1 ROT R ROT POS
OR        M12806	// T)R_1st ROT R ROT POS PLS
OR        M03111	// R_1-1 ROT R ROT POS ->
AND       T0711	// R_1-1 ROT R READY 2s
OUT       M03111	// R_1-1 ROT R ROT POS ->
; L183
LOAD      M12580	// R_1st MAND CYCLE RUN
AND       M12518	// 06_R move back pos
AND NOT   M04112	// R_1-1 ROT R BACK POS
OR        M1280A	// T)R_1st ROT R BACK POS ->
OR        M03112	// R_1-1 ROT R BACK POS ->
AND       T0711	// R_1-1 ROT R READY 2s
OUT       M03112	// R_1-1 ROT R BACK POS ->
// ======================== 13_R_1st ROTATE Y ==========================
; L187
LOAD      M12580	// R_1st MAND CYCLE RUN
AND NOT   M04130	// R_1st ROT Y 1st POS
LOAD      M1280D	// T)R_1st ROT Y 1st POS ->
AND       M01632	// R_1st ROT Y HOME COMPLETE
OR LOAD
OR        M03130	// R_1st ROT Y 1st POS ->
AND       T0713	// R_1st ROT Y READY 2s
OUT       M03130	// R_1st ROT Y 1st POS ->
; L190
LOAD      M12580	// R_1st MAND CYCLE RUN
AND NOT   M04131	// R_1st ROT Y 2nd POS
OR        M1280F	// T)R_1st ROT Y 2nd POS ->
OR        M03131	// R_1st ROT Y 2nd POS ->
AND       T0713	// R_1st ROT Y READY 2s
AND       F0009A
OUT       M03131	// R_1st ROT Y 2nd POS ->
; L193
END

PROGRAM 17_R_2nd_MAND (task: ½ºÄµ ÇÁ·Î±×·¥)

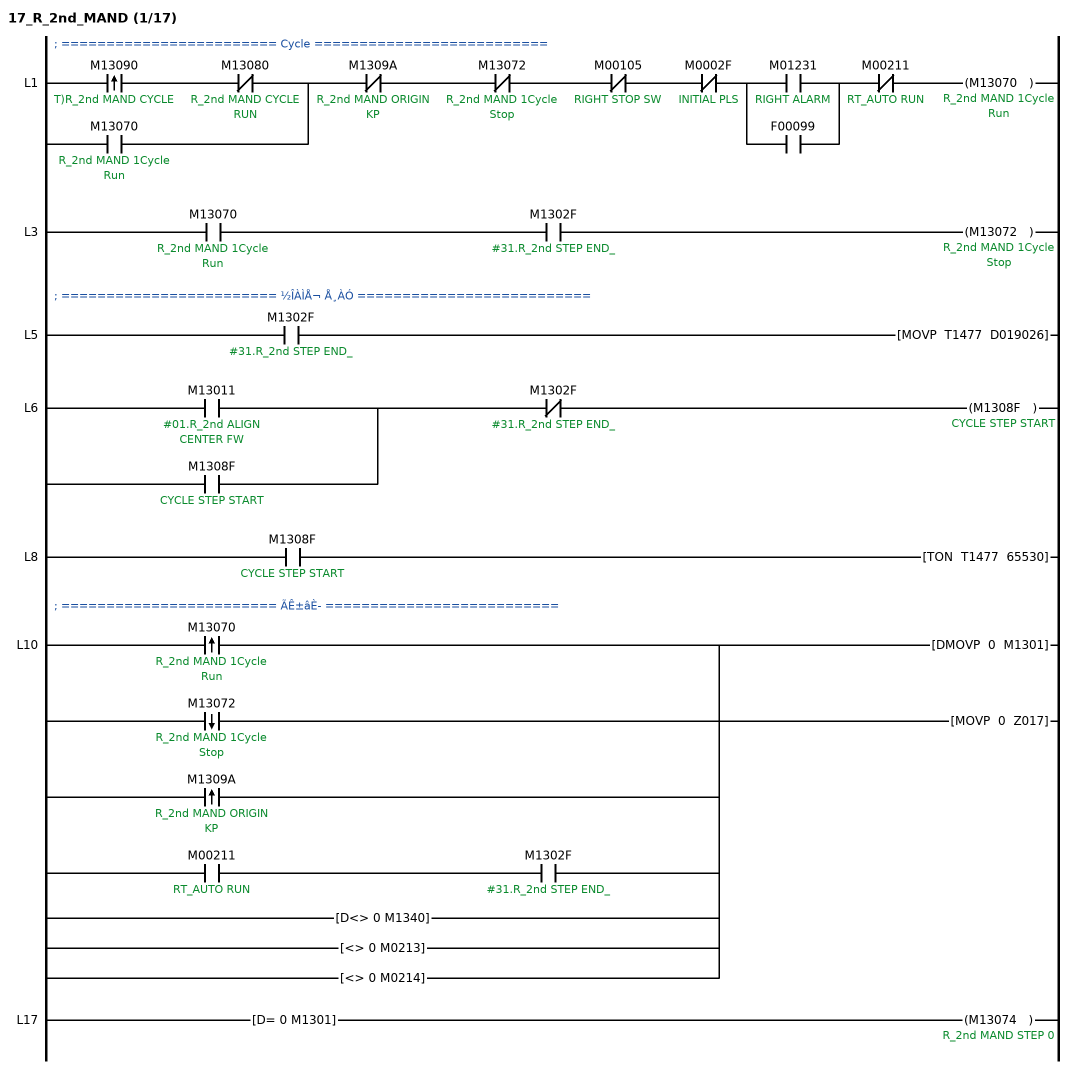
// ======================== Cycle ==========================
; L1
LOADP     M13090	// T)R_2nd MAND CYCLE
AND NOT   M13080	// R_2nd MAND CYCLE RUN
OR        M13070	// R_2nd MAND 1Cycle Run
AND NOT   M1309A	// R_2nd MAND ORIGIN KP
AND NOT   M13072	// R_2nd MAND 1Cycle Stop
AND NOT   M00105	// RIGHT STOP SW
AND NOT   M0002F	// INITIAL PLS
LOAD      M01231	// RIGHT ALARM
OR        F00099
AND LOAD
AND NOT   M00211	// RT_AUTO RUN
OUT       M13070	// R_2nd MAND 1Cycle Run
; L3
LOAD      M13070	// R_2nd MAND 1Cycle Run
AND       M1302F	// #31.R_2nd STEP END_
OUT       M13072	// R_2nd MAND 1Cycle Stop
// ======================== ½ÎÀÌÅ¬ Å¸ÀÓ ==========================
; L5
LOAD      M1302F	// #31.R_2nd STEP END_
MOVP      T1477 D019026
; L6
LOAD      M13011	// #01.R_2nd ALIGN CENTER FW
OR        M1308F	// CYCLE STEP START
AND NOT   M1302F	// #31.R_2nd STEP END_
OUT       M1308F	// CYCLE STEP START
; L8
LOAD      M1308F	// CYCLE STEP START
TON       T1477 65530
// ======================== ÃÊ±âÈ­ ==========================
; L10
LOADP     M13070	// R_2nd MAND 1Cycle Run
ORN       M13072	// R_2nd MAND 1Cycle Stop
ORP       M1309A	// R_2nd MAND ORIGIN KP
LOAD      M00211	// RT_AUTO RUN
AND       M1302F	// #31.R_2nd STEP END_
OR LOAD
ORD<>     0 M1340
OR<>      0 M0213
OR<>      0 M0214
DMOVP     0 M1301
MOVP      0 Z017
; L17
LOADD=    0 M1301
OUT       M13074	// R_2nd MAND STEP 0

